QRS_NEXT_CUT()
PTP {E1 35817.312,E2 35817.312}
PTP {X 0,Y 759.87,A -85,B 0,C 180,E1 35817.312,E2 35817.312,E3 0,E4 0,E5 0,E6 0}
QRS_SPEED_INIT()
LIN {X 0,Y 759.87,Z 1164.5,A -85,B 0,C 180,E1 35817.312,E2 35817.312,E3 0,E4 0,E5 0,E6 0} C_VEL
LIN {X 0,Y 759.87,Z 412.653,A -85,B 0,C 180,E1 35817.312,E2 35817.312} C_VEL
LIN {X 0,Y 759.87,Z 404.575,A -85,B 0,C 180,E1 35817.312,E2 35817.312} C_VEL
LIN {X 0,Y 759.853,Z 402.575,A -85,B 0,C 180,E1 35817.162,E2 35817.162} C_VEL
LIN {X 0,Y 759.833,Z 402.574,A -85,B 0,C 180,E1 35814.715,E2 35814.715} C_VEL
LIN {X 0,Y 759.853,Z 402.572,A -85,B 0,C 180,E1 35812.255,E2 35812.255} C_VEL
LIN {X 0,Y 759.868,Z 402.576,A -85,B 0,C 180,E1 35809.231,E2 35809.231} C_VEL
LIN {X 0,Y 759.827,Z 402.575,A -85,B 0,C 180,E1 35806.763,E2 35806.763} C_VEL
LIN {X 0,Y 759.822,Z 402.575,A -85,B 0,C 180,E1 35804.506,E2 35804.506} C_VEL
LIN {X 0,Y 759.836,Z 402.574,A -85,B 0,C 180,E1 35802.145,E2 35802.145} C_VEL
LIN {X 0,Y 759.892,Z 402.577,A -85,B 0,C 180,E1 35799.27,E2 35799.27} C_VEL
LIN {X 0,Y 759.819,Z 402.576,A -85,B 0,C 180,E1 35796.665,E2 35796.665} C_VEL
LIN {X 0,Y 759.81,Z 402.576,A -85,B 0,C 180,E1 35794.428,E2 35794.428} C_VEL
LIN {X 0,Y 759.809,Z 402.576,A -85,B 0,C 180,E1 35792.234,E2 35792.234} C_VEL
LIN {X 0,Y 759.824,Z 402.577,A -85,B 0,C 180,E1 35789.909,E2 35789.909} C_VEL
LIN {X 0,Y 759.858,Z 402.577,A -85,B 0,C 180,E1 35786.953,E2 35786.953} C_VEL
LIN {X 0,Y 759.813,Z 402.576,A -85,B 0,C 180,E1 35784.525,E2 35784.525} C_VEL
LIN {X 0,Y 759.809,Z 402.577,A -85,B 0,C 180,E1 35782.366,E2 35782.366} C_VEL
LIN {X 0,Y 759.807,Z 402.577,A -85,B 0,C 180,E1 35780.223,E2 35780.223} C_VEL
LIN {X 0,Y 759.811,Z 402.576,A -85,B 0,C 180,E1 35778.033,E2 35778.033} C_VEL
LIN {X 0,Y 759.832,Z 402.577,A -85,B 0,C 180,E1 35775.672,E2 35775.672} C_VEL
LIN {X 0,Y 759.881,Z 402.574,A -85,B 0,C 180,E1 35772.756,E2 35772.756} C_VEL
LIN {X 0,Y 759.828,Z 402.575,A -85,B 0,C 180,E1 35770.248,E2 35770.248} C_VEL
LIN {X 0,Y 759.822,Z 402.575,A -85,B 0,C 180,E1 35767.919,E2 35767.919} C_VEL
LIN {X 0,Y 759.838,Z 402.576,A -85,B 0,C 180,E1 35765.566,E2 35765.566} C_VEL
LIN {X 0,Y 759.89,Z 402.904,A -85,B 0,C 180,E1 35765.147,E2 35765.147} C_VEL
LIN {X 0,Y 759.915,Z 438.12,A -85,B 0,C 180,E1 35762.827,E2 35762.827} C_VEL
LIN {X 0,Y 759.889,Z 482.271,A -85,B 0,C 180,E1 35760.023,E2 35760.023} C_VEL
LIN {X 0,Y 759.879,Z 498.982,A -85,B 0,C 180,E1 35758.995,E2 35758.995} C_VEL
LIN {X 0,Y 759.908,Z 754.621,A -85,B 0,C 180,E1 35756.312,E2 35756.312} C_VEL
LIN {X 0,Y 759.901,Z 846.139,A -85,B 0,C 180,E1 35755.349,E2 35755.349} C_VEL
LIN {X 0,Y 759.915,Z 869.708,A -85,B 0,C 180,E1 35754.962,E2 35754.962} C_VEL
LIN {X 0,Y 759.917,Z 889.343,A -85,B 0,C 180,E1 35754.528,E2 35754.528} C_VEL
LIN {X 0,Y 759.899,Z 912.803,A -85,B 0,C 180,E1 35753.865,E2 35753.865} C_VEL
LIN {X 0,Y 759.919,Z 931.783,A -85,B 0,C 180,E1 35753.209,E2 35753.209} C_VEL
LIN {X 0,Y 759.917,Z 953.84,A -85,B 0,C 180,E1 35752.3,E2 35752.3} C_VEL
LIN {X 0,Y 759.913,Z 972.967,A -85,B 0,C 180,E1 35751.375,E2 35751.375} C_VEL
LIN {X 0,Y 759.916,Z 992.86,A -85,B 0,C 180,E1 35750.255,E2 35750.255} C_VEL
LIN {X 0,Y 759.91,Z 1011.008,A -85,B 0,C 180,E1 35749.085,E2 35749.085} C_VEL
LIN {X 0,Y 759.908,Z 1028.563,A -85,B 0,C 180,E1 35747.774,E2 35747.774} C_VEL
LIN {X 0,Y 759.919,Z 1045.141,A -85,B 0,C 180,E1 35746.355,E2 35746.355} C_VEL
LIN {X 0,Y 759.902,Z 1059.575,A -85,B 0,C 180,E1 35744.946,E2 35744.946} C_VEL
LIN {X 0,Y 759.901,Z 1072.566,A -85,B 0,C 180,E1 35743.468,E2 35743.468} C_VEL
LIN {X 0,Y 759.915,Z 1084.432,A -85,B 0,C 180,E1 35741.922,E2 35741.922} C_VEL
LIN {X 0,Y 759.908,Z 1094.369,A -85,B 0,C 180,E1 35740.385,E2 35740.385} C_VEL
LIN {X 0,Y 759.894,Z 1103.565,A -85,B 0,C 180,E1 35738.703,E2 35738.703} C_VEL
LIN {X 0,Y 759.917,Z 1110.573,A -85,B 0,C 180,E1 35737.105,E2 35737.105} C_VEL
LIN {X 0,Y 759.896,Z 1116.604,A -85,B 0,C 180,E1 35735.361,E2 35735.361} C_VEL
LIN {X 0,Y 759.895,Z 1120.521,A -85,B 0,C 180,E1 35733.772,E2 35733.772} C_VEL
LIN {X 0,Y 759.915,Z 1123.316,A -85,B 0,C 180,E1 35732.036,E2 35732.036} C_VEL
LIN {X 0,Y 759.894,Z 1124.382,A -85,B 0,C 180,E1 35730.377,E2 35730.377} C_VEL
LIN {X 0,Y 759.893,Z 1123.929,A -85,B 0,C 180,E1 35728.567,E2 35728.567} C_VEL
LIN {X 0,Y 759.908,Z 1122.072,A -85,B 0,C 180,E1 35726.983,E2 35726.983} C_VEL
LIN {X 0,Y 759.892,Z 1118.285,A -85,B 0,C 180,E1 35725.169,E2 35725.169} C_VEL
LIN {X 0,Y 759.9,Z 1113.46,A -85,B 0,C 180,E1 35723.578,E2 35723.578} C_VEL
LIN {X 0,Y 759.912,Z 1106.463,A -85,B 0,C 180,E1 35721.83,E2 35721.83} C_VEL
LIN {X 0,Y 759.893,Z 1098.847,A -85,B 0,C 180,E1 35720.304,E2 35720.304} C_VEL
LIN {X 0,Y 759.9,Z 1088.594,A -85,B 0,C 180,E1 35718.605,E2 35718.605} C_VEL
LIN {X 0,Y 759.911,Z 1078.231,A -85,B 0,C 180,E1 35717.152,E2 35717.152} C_VEL
LIN {X 0,Y 759.917,Z 1065.021,A -85,B 0,C 180,E1 35715.564,E2 35715.564} C_VEL
LIN {X 0,Y 759.903,Z 1051.164,A -85,B 0,C 180,E1 35714.116,E2 35714.116} C_VEL
LIN {X 0,Y 759.905,Z 1035.427,A -85,B 0,C 180,E1 35712.7,E2 35712.7} C_VEL
LIN {X 0,Y 759.91,Z 1018.024,A -85,B 0,C 180,E1 35711.331,E2 35711.331} C_VEL
LIN {X 0,Y 759.91,Z 1000.339,A -85,B 0,C 180,E1 35710.115,E2 35710.115} C_VEL
LIN {X 0,Y 759.911,Z 981.35,A -85,B 0,C 180,E1 35708.988,E2 35708.988} C_VEL
LIN {X 0,Y 759.915,Z 961.832,A -85,B 0,C 180,E1 35707.976,E2 35707.976} C_VEL
LIN {X 0,Y 759.918,Z 941.464,A -85,B 0,C 180,E1 35707.081,E2 35707.081} C_VEL
LIN {X 0,Y 759.902,Z 920.345,A -85,B 0,C 180,E1 35706.289,E2 35706.289} C_VEL
LIN {X 0,Y 759.918,Z 899.782,A -85,B 0,C 180,E1 35705.659,E2 35705.659} C_VEL
LIN {X 0,Y 759.909,Z 878.291,A -85,B 0,C 180,E1 35705.119,E2 35705.119} C_VEL
LIN {X 0,Y 759.91,Z 857.163,A -85,B 0,C 180,E1 35704.725,E2 35704.725} C_VEL
LIN {X 0,Y 759.899,Z 835.535,A -85,B 0,C 180,E1 35704.431,E2 35704.431} C_VEL
LIN {X 0,Y 759.87,Z 588.613,A -85,B 0,C 180,E1 35701.868,E2 35701.868} C_VEL
LIN {X 0,Y 759.879,Z 498.825,A -85,B 0,C 180,E1 35700.91,E2 35700.91} C_VEL
LIN {X 0,Y 759.891,Z 459.664,A -85,B 0,C 180,E1 35698.461,E2 35698.461} C_VEL
LIN {X 0,Y 759.918,Z 417.942,A -85,B 0,C 180,E1 35695.771,E2 35695.771} C_VEL
LIN {X 0,Y 759.892,Z 402.857,A -85,B 0,C 180,E1 35694.756,E2 35694.756} C_VEL
LIN {X 0,Y 759.884,Z 402.572,A -85,B 0,C 180,E1 35693.386,E2 35693.386} C_VEL
LIN {X 0,Y 759.854,Z 402.576,A -85,B 0,C 180,E1 35690.439,E2 35690.439} C_VEL
LIN {X 0,Y 759.827,Z 402.575,A -85,B 0,C 180,E1 35688.031,E2 35688.031} C_VEL
LIN {X 0,Y 759.831,Z 402.573,A -85,B 0,C 180,E1 35685.672,E2 35685.672} C_VEL
LIN {X 0,Y 759.911,Z 402.574,A -85,B 0,C 180,E1 35682.968,E2 35682.968} C_VEL
LIN {X 0,Y 759.828,Z 402.576,A -85,B 0,C 180,E1 35680.132,E2 35680.132} C_VEL
LIN {X 0,Y 759.815,Z 402.576,A -85,B 0,C 180,E1 35677.853,E2 35677.853} C_VEL
LIN {X 0,Y 759.812,Z 402.575,A -85,B 0,C 180,E1 35675.66,E2 35675.66} C_VEL
LIN {X 0,Y 759.822,Z 402.576,A -85,B 0,C 180,E1 35673.372,E2 35673.372} C_VEL
LIN {X 0,Y 759.894,Z 402.578,A -85,B 0,C 180,E1 35670.525,E2 35670.525} C_VEL
LIN {X 0,Y 759.812,Z 402.577,A -85,B 0,C 180,E1 35667.936,E2 35667.936} C_VEL
LIN {X 0,Y 759.802,Z 402.577,A -85,B 0,C 180,E1 35665.65,E2 35665.65} C_VEL
LIN {X 0,Y 759.805,Z 402.577,A -85,B 0,C 180,E1 35663.5,E2 35663.5} C_VEL
LIN {X 0,Y 759.812,Z 402.577,A -85,B 0,C 180,E1 35661.297,E2 35661.297} C_VEL
LIN {X 0,Y 759.891,Z 402.577,A -85,B 0,C 180,E1 35658.648,E2 35658.648} C_VEL
LIN {X 0,Y 759.833,Z 402.575,A -85,B 0,C 180,E1 35655.807,E2 35655.807} C_VEL
LIN {X 0,Y 759.819,Z 402.575,A -85,B 0,C 180,E1 35653.468,E2 35653.468} C_VEL
LIN {X 0,Y 759.822,Z 402.575,A -85,B 0,C 180,E1 35651.231,E2 35651.231} C_VEL
LIN {X 0,Y 759.856,Z 402.576,A -85,B 0,C 180,E1 35648.78,E2 35648.78} C_VEL
LIN {X 0,Y 759.856,Z 402.573,A -85,B 0,C 180,E1 35645.74,E2 35645.74} C_VEL
LIN {X 0,Y 759.832,Z 402.573,A -85,B 0,C 180,E1 35643.319,E2 35643.319} C_VEL
LIN {X 0,Y 759.841,Z 402.575,A -85,B 0,C 180,E1 35640.905,E2 35640.905} C_VEL
LIN {X 0,Y 759.917,Z 402.575,A -85,B 0,C 180,E1 35638.19,E2 35638.19} C_VEL
LIN {X 0,Y 759.851,Z 402.571,A -85,B 0,C 180,E1 35635.396,E2 35635.396} C_VEL
LIN {X 0,Y 759.842,Z 402.573,A -85,B 0,C 180,E1 35632.97,E2 35632.97} C_VEL
LIN {X 0,Y 759.901,Z 402.577,A -85,B 0,C 180,E1 35630.304,E2 35630.304} C_VEL
LIN {X 0,Y 759.871,Z 402.569,A -85,B 0,C 180,E1 35627.383,E2 35627.383} C_VEL
LIN {X 0,Y 759.851,Z 402.573,A -85,B 0,C 180,E1 35624.819,E2 35624.819} C_VEL
LIN {X 0,Y 759.908,Z 402.578,A -85,B 0,C 180,E1 35622.147,E2 35622.147} C_VEL
LIN {X 0,Y 759.874,Z 402.569,A -85,B 0,C 180,E1 35619.189,E2 35619.189} C_VEL
LIN {X 0,Y 759.866,Z 402.573,A -85,B 0,C 180,E1 35616.516,E2 35616.516} C_VEL
LIN {X 0,Y 759.909,Z 402.572,A -85,B 0,C 180,E1 35613.761,E2 35613.761} C_VEL
LIN {X 0,Y 759.873,Z 402.568,A -85,B 0,C 180,E1 35610.951,E2 35610.951} C_VEL
LIN {X 0,Y 759.887,Z 402.575,A -85,B 0,C 180,E1 35608.216,E2 35608.216} C_VEL
LIN {X 0,Y 759.917,Z 402.564,A -85,B 0,C 180,E1 35605.268,E2 35605.268} C_VEL
LIN {X 0,Y 759.872,Z 402.572,A -85,B 0,C 180,E1 35602.465,E2 35602.465} C_VEL
LIN {X 0,Y 759.911,Z 402.575,A -85,B 0,C 180,E1 35599.744,E2 35599.744} C_VEL
LIN {X 0,Y 759.892,Z 402.566,A -85,B 0,C 180,E1 35596.801,E2 35596.801} C_VEL
LIN {X 0,Y 759.906,Z 402.576,A -85,B 0,C 180,E1 35593.903,E2 35593.903} C_VEL
LIN {X 0,Y 759.908,Z 402.565,A -85,B 0,C 180,E1 35590.835,E2 35590.835} C_VEL
LIN {X 0,Y 759.905,Z 402.577,A -85,B 0,C 180,E1 35587.862,E2 35587.862} C_VEL
LIN {X 0,Y 759.901,Z 402.734,A -85,B 0,C 180,E1 35585.893,E2 35585.893} C_VEL
LIN {X 0,Y 759.916,Z 406.955,A -85,B 0,C 180,E1 35585.594,E2 35585.594} C_VEL
LIN {X 0,Y 759.899,Z 450.794,A -85,B 0,C 180,E1 35582.913,E2 35582.913} C_VEL
LIN {X 0,Y 759.909,Z 452.682,A -85,B 0,C 180,E1 35582.815,E2 35582.815} C_VEL
LIN {X 0,Y 759.892,Z 704.216,A -85,B 0,C 180,E1 35580.08,E2 35580.08} C_VEL
LIN {X 0,Y 759.92,Z 841.979,A -85,B 0,C 180,E1 35578.595,E2 35578.595} C_VEL
LIN {X 0,Y 759.894,Z 866.292,A -85,B 0,C 180,E1 35578.211,E2 35578.211} C_VEL
LIN {X 0,Y 759.9,Z 887.681,A -85,B 0,C 180,E1 35577.742,E2 35577.742} C_VEL
LIN {X 0,Y 759.897,Z 907.094,A -85,B 0,C 180,E1 35577.221,E2 35577.221} C_VEL
LIN {X 0,Y 759.919,Z 929.734,A -85,B 0,C 180,E1 35576.491,E2 35576.491} C_VEL
LIN {X 0,Y 759.916,Z 951.248,A -85,B 0,C 180,E1 35575.652,E2 35575.652} C_VEL
LIN {X 0,Y 759.913,Z 970.659,A -85,B 0,C 180,E1 35574.783,E2 35574.783} C_VEL
LIN {X 0,Y 759.91,Z 993.058,A -85,B 0,C 180,E1 35573.62,E2 35573.62} C_VEL
LIN {X 0,Y 759.92,Z 1011.704,A -85,B 0,C 180,E1 35572.513,E2 35572.513} C_VEL
LIN {X 0,Y 759.906,Z 1031.522,A -85,B 0,C 180,E1 35571.173,E2 35571.173} C_VEL
LIN {X 0,Y 759.916,Z 1048.884,A -85,B 0,C 180,E1 35569.845,E2 35569.845} C_VEL
LIN {X 0,Y 759.917,Z 1065.39,A -85,B 0,C 180,E1 35568.409,E2 35568.409} C_VEL
LIN {X 0,Y 759.895,Z 1079.946,A -85,B 0,C 180,E1 35566.985,E2 35566.985} C_VEL
LIN {X 0,Y 759.899,Z 1094.876,A -85,B 0,C 180,E1 35565.312,E2 35565.312} C_VEL
LIN {X 0,Y 759.905,Z 1106.572,A -85,B 0,C 180,E1 35563.815,E2 35563.815} C_VEL
LIN {X 0,Y 759.9,Z 1118.785,A -85,B 0,C 180,E1 35561.999,E2 35561.999} C_VEL
LIN {X 0,Y 759.907,Z 1127.555,A -85,B 0,C 180,E1 35560.462,E2 35560.462} C_VEL
LIN {X 0,Y 759.888,Z 1136.073,A -85,B 0,C 180,E1 35558.704,E2 35558.704} C_VEL
LIN {X 0,Y 759.918,Z 1142.726,A -85,B 0,C 180,E1 35556.953,E2 35556.953} C_VEL
LIN {X 0,Y 759.883,Z 1147.51,A -85,B 0,C 180,E1 35555.361,E2 35555.361} C_VEL
LIN {X 0,Y 759.919,Z 1151.559,A -85,B 0,C 180,E1 35553.47,E2 35553.47} C_VEL
LIN {X 0,Y 759.902,Z 1153.63,A -85,B 0,C 180,E1 35551.81,E2 35551.81} C_VEL
LIN {X 0,Y 759.92,Z 1154.5,A -85,B 0,C 180,E1 35550,E2 35550} C_VEL
LIN {X 0,Y 759.902,Z 1153.63,A -85,B 0,C 180,E1 35548.19,E2 35548.19} C_VEL
LIN {X 0,Y 759.919,Z 1151.559,A -85,B 0,C 180,E1 35546.53,E2 35546.53} C_VEL
LIN {X 0,Y 759.883,Z 1147.51,A -85,B 0,C 180,E1 35544.639,E2 35544.639} C_VEL
LIN {X 0,Y 759.918,Z 1142.726,A -85,B 0,C 180,E1 35543.047,E2 35543.047} C_VEL
LIN {X 0,Y 759.889,Z 1135.729,A -85,B 0,C 180,E1 35541.22,E2 35541.22} C_VEL
LIN {X 0,Y 759.907,Z 1127.555,A -85,B 0,C 180,E1 35539.538,E2 35539.538} C_VEL
LIN {X 0,Y 759.9,Z 1118.785,A -85,B 0,C 180,E1 35538.001,E2 35538.001} C_VEL
LIN {X 0,Y 759.904,Z 1106.265,A -85,B 0,C 180,E1 35536.144,E2 35536.144} C_VEL
LIN {X 0,Y 759.9,Z 1094.679,A -85,B 0,C 180,E1 35534.664,E2 35534.664} C_VEL
LIN {X 0,Y 759.896,Z 1079.169,A -85,B 0,C 180,E1 35532.937,E2 35532.937} C_VEL
LIN {X 0,Y 759.914,Z 1064.539,A -85,B 0,C 180,E1 35531.512,E2 35531.512} C_VEL
LIN {X 0,Y 759.913,Z 1046.484,A -85,B 0,C 180,E1 35529.965,E2 35529.965} C_VEL
LIN {X 0,Y 759.91,Z 1029.578,A -85,B 0,C 180,E1 35528.684,E2 35528.684} C_VEL
LIN {X 0,Y 759.918,Z 1009.719,A -85,B 0,C 180,E1 35527.364,E2 35527.364} C_VEL
LIN {X 0,Y 759.91,Z 990.876,A -85,B 0,C 180,E1 35526.257,E2 35526.257} C_VEL
LIN {X 0,Y 759.913,Z 969.006,A -85,B 0,C 180,E1 35525.14,E2 35525.14} C_VEL
LIN {X 0,Y 759.917,Z 950.063,A -85,B 0,C 180,E1 35524.299,E2 35524.299} C_VEL
LIN {X 0,Y 759.915,Z 927.316,A -85,B 0,C 180,E1 35523.425,E2 35523.425} C_VEL
LIN {X 0,Y 759.899,Z 906.002,A -85,B 0,C 180,E1 35522.748,E2 35522.748} C_VEL
LIN {X 0,Y 759.898,Z 886.062,A -85,B 0,C 180,E1 35522.218,E2 35522.218} C_VEL
LIN {X 0,Y 759.898,Z 861.401,A -85,B 0,C 180,E1 35521.701,E2 35521.701} C_VEL
LIN {X 0,Y 759.92,Z 840.266,A -85,B 0,C 180,E1 35521.383,E2 35521.383} C_VEL
LIN {X 0,Y 759.859,Z 578.286,A -85,B 0,C 180,E1 35518.562,E2 35518.562} C_VEL
LIN {X 0,Y 759.907,Z 452.293,A -85,B 0,C 180,E1 35517.172,E2 35517.172} C_VEL
LIN {X 0,Y 759.92,Z 408.959,A -85,B 0,C 180,E1 35514.531,E2 35514.531} C_VEL
LIN {X 0,Y 759.902,Z 402.854,A -85,B 0,C 180,E1 35514.128,E2 35514.128} C_VEL
LIN {X 0,Y 759.903,Z 402.572,A -85,B 0,C 180,E1 35512.467,E2 35512.467} C_VEL
LIN {X 0,Y 759.882,Z 402.572,A -85,B 0,C 180,E1 35509.747,E2 35509.747} C_VEL
LIN {X 0,Y 759.909,Z 402.565,A -85,B 0,C 180,E1 35506.909,E2 35506.909} C_VEL
LIN {X 0,Y 759.896,Z 402.575,A -85,B 0,C 180,E1 35503.965,E2 35503.965} C_VEL
LIN {X 0,Y 759.9,Z 402.565,A -85,B 0,C 180,E1 35501.065,E2 35501.065} C_VEL
LIN {X 0,Y 759.908,Z 402.577,A -85,B 0,C 180,E1 35498.01,E2 35498.01} C_VEL
LIN {X 0,Y 759.877,Z 402.568,A -85,B 0,C 180,E1 35495.194,E2 35495.194} C_VEL
LIN {X 0,Y 759.906,Z 402.57,A -85,B 0,C 180,E1 35492.38,E2 35492.38} C_VEL
LIN {X 0,Y 759.873,Z 402.573,A -85,B 0,C 180,E1 35489.566,E2 35489.566} C_VEL
LIN {X 0,Y 759.888,Z 402.567,A -85,B 0,C 180,E1 35486.829,E2 35486.829} C_VEL
LIN {X 0,Y 759.901,Z 402.577,A -85,B 0,C 180,E1 35483.826,E2 35483.826} C_VEL
LIN {X 0,Y 759.859,Z 402.571,A -85,B 0,C 180,E1 35481.134,E2 35481.134} C_VEL
LIN {X 0,Y 759.912,Z 402.566,A -85,B 0,C 180,E1 35478.409,E2 35478.409} C_VEL
LIN {X 0,Y 759.873,Z 402.575,A -85,B 0,C 180,E1 35475.493,E2 35475.493} C_VEL
LIN {X 0,Y 759.852,Z 402.571,A -85,B 0,C 180,E1 35472.927,E2 35472.927} C_VEL
LIN {X 0,Y 759.917,Z 402.568,A -85,B 0,C 180,E1 35470.193,E2 35470.193} C_VEL
LIN {X 0,Y 759.863,Z 402.575,A -85,B 0,C 180,E1 35467.333,E2 35467.333} C_VEL
LIN {X 0,Y 759.844,Z 402.572,A -85,B 0,C 180,E1 35464.831,E2 35464.831} C_VEL
LIN {X 0,Y 759.895,Z 402.569,A -85,B 0,C 180,E1 35462.187,E2 35462.187} C_VEL
LIN {X 0,Y 759.86,Z 402.576,A -85,B 0,C 180,E1 35459.246,E2 35459.246} C_VEL
LIN {X 0,Y 759.853,Z 402.575,A -85,B 0,C 180,E1 35457.162,E2 35457.162} C_VEL
LIN {X 0,Y 758.828,Z 402.701,A -85,B 0,C 180,E1 35456.581,E2 35456.581} C_VEL
LIN {X 0,Y 752.415,Z 403.5,A -85,B 0,C 180,E1 35454.954,E2 35454.954} C_VEL
LIN {X 0,Y 751.899,Z 403.562,A -85,B 0,C 180,E1 35454.531,E2 35454.531} C_VEL
LIN {X 0,Y 751.971,Z 403.56,A -85,B 0,C 180,E1 35451.82,E2 35451.82} C_VEL
LIN {X 0,Y 751.9,Z 403.564,A -85,B 0,C 180,E1 35448.96,E2 35448.96} C_VEL
LIN {X 0,Y 751.885,Z 403.564,A -85,B 0,C 180,E1 35446.621,E2 35446.621} C_VEL
LIN {X 0,Y 751.89,Z 403.563,A -85,B 0,C 180,E1 35444.324,E2 35444.324} C_VEL
LIN {X 0,Y 751.977,Z 403.563,A -85,B 0,C 180,E1 35441.551,E2 35441.551} C_VEL
LIN {X 0,Y 751.888,Z 403.565,A -85,B 0,C 180,E1 35438.784,E2 35438.784} C_VEL
LIN {X 0,Y 751.874,Z 403.565,A -85,B 0,C 180,E1 35436.487,E2 35436.487} C_VEL
LIN {X 0,Y 751.872,Z 403.565,A -85,B 0,C 180,E1 35434.308,E2 35434.308} C_VEL
LIN {X 0,Y 751.883,Z 403.565,A -85,B 0,C 180,E1 35432.002,E2 35432.002} C_VEL
LIN {X 0,Y 751.958,Z 403.566,A -85,B 0,C 180,E1 35429.205,E2 35429.205} C_VEL
LIN {X 0,Y 751.87,Z 403.566,A -85,B 0,C 180,E1 35426.495,E2 35426.495} C_VEL
LIN {X 0,Y 751.865,Z 403.563,A -85,B 0,C 180,E1 35424.28,E2 35424.28} C_VEL
LIN {X 0,Y 751.869,Z 403.566,A -85,B 0,C 180,E1 35422.057,E2 35422.057} C_VEL
LIN {X 0,Y 751.888,Z 403.566,A -85,B 0,C 180,E1 35419.736,E2 35419.736} C_VEL
LIN {X 0,Y 751.93,Z 403.565,A -85,B 0,C 180,E1 35416.778,E2 35416.778} C_VEL
LIN {X 0,Y 751.882,Z 403.562,A -85,B 0,C 180,E1 35414.281,E2 35414.281} C_VEL
LIN {X 0,Y 751.879,Z 403.565,A -85,B 0,C 180,E1 35411.979,E2 35411.979} C_VEL
LIN {X 0,Y 751.901,Z 403.565,A -85,B 0,C 180,E1 35409.567,E2 35409.567} C_VEL
LIN {X 0,Y 751.95,Z 403.563,A -85,B 0,C 180,E1 35406.659,E2 35406.659} C_VEL
LIN {X 0,Y 751.93,Z 403.764,A -85,B 0,C 180,E1 35405.529,E2 35405.529} C_VEL
LIN {X 0,Y 752.835,Z 407.065,A -85,B 0,C 180,E1 35405.232,E2 35405.232} C_VEL
LIN {X 0,Y 752.698,Z 447.098,A -85,B 0,C 180,E1 35402.598,E2 35402.598} C_VEL
LIN {X 0,Y 752.547,Z 488.811,A -85,B 0,C 180,E1 35399.933,E2 35399.933} C_VEL
LIN {X 0,Y 752.641,Z 499.389,A -85,B 0,C 180,E1 35399.293,E2 35399.293} C_VEL
LIN {X 0,Y 752.884,Z 507.669,A -85,B 0,C 180,E1 35399.189,E2 35399.189} C_VEL
LIN {X 0,Y 752.725,Z 771.08,A -85,B 0,C 180,E1 35396.412,E2 35396.412} C_VEL
LIN {X 0,Y 752.664,Z 846.932,A -85,B 0,C 180,E1 35395.601,E2 35395.601} C_VEL
LIN {X 0,Y 752.63,Z 870.129,A -85,B 0,C 180,E1 35395.213,E2 35395.213} C_VEL
LIN {X 0,Y 752.589,Z 890.661,A -85,B 0,C 180,E1 35394.751,E2 35394.751} C_VEL
LIN {X 0,Y 752.497,Z 913.406,A -85,B 0,C 180,E1 35394.096,E2 35394.096} C_VEL
LIN {X 0,Y 752.459,Z 934.151,A -85,B 0,C 180,E1 35393.365,E2 35393.365} C_VEL
LIN {X 0,Y 752.373,Z 955.428,A -85,B 0,C 180,E1 35392.463,E2 35392.463} C_VEL
LIN {X 0,Y 752.305,Z 975.361,A -85,B 0,C 180,E1 35391.48,E2 35391.48} C_VEL
LIN {X 0,Y 752.229,Z 994.993,A -85,B 0,C 180,E1 35390.34,E2 35390.34} C_VEL
LIN {X 0,Y 752.153,Z 1014.194,A -85,B 0,C 180,E1 35389.058,E2 35389.058} C_VEL
LIN {X 0,Y 752.102,Z 1031.589,A -85,B 0,C 180,E1 35387.725,E2 35387.725} C_VEL
LIN {X 0,Y 752.051,Z 1047.695,A -85,B 0,C 180,E1 35386.292,E2 35386.292} C_VEL
LIN {X 0,Y 751.998,Z 1063.127,A -85,B 0,C 180,E1 35384.712,E2 35384.712} C_VEL
LIN {X 0,Y 751.962,Z 1076.4,A -85,B 0,C 180,E1 35383.143,E2 35383.143} C_VEL
LIN {X 0,Y 751.93,Z 1087.547,A -85,B 0,C 180,E1 35381.583,E2 35381.583} C_VEL
LIN {X 0,Y 751.922,Z 1097.557,A -85,B 0,C 180,E1 35379.955,E2 35379.955} C_VEL
LIN {X 0,Y 751.916,Z 1105.693,A -85,B 0,C 180,E1 35378.334,E2 35378.334} C_VEL
LIN {X 0,Y 751.893,Z 1112.824,A -85,B 0,C 180,E1 35376.592,E2 35376.592} C_VEL
LIN {X 0,Y 751.907,Z 1117.838,A -85,B 0,C 180,E1 35374.959,E2 35374.959} C_VEL
LIN {X 0,Y 751.903,Z 1121.716,A -85,B 0,C 180,E1 35373.202,E2 35373.202} C_VEL
LIN {X 0,Y 751.89,Z 1123.783,A -85,B 0,C 180,E1 35371.524,E2 35371.524} C_VEL
LIN {X 0,Y 751.903,Z 1124.453,A -85,B 0,C 180,E1 35369.771,E2 35369.771} C_VEL
LIN {X 0,Y 751.906,Z 1123.529,A -85,B 0,C 180,E1 35368.095,E2 35368.095} C_VEL
LIN {X 0,Y 751.895,Z 1120.867,A -85,B 0,C 180,E1 35366.264,E2 35366.264} C_VEL
LIN {X 0,Y 751.906,Z 1117.053,A -85,B 0,C 180,E1 35364.659,E2 35364.659} C_VEL
LIN {X 0,Y 751.915,Z 1110.93,A -85,B 0,C 180,E1 35362.819,E2 35362.819} C_VEL
LIN {X 0,Y 751.902,Z 1104.335,A -85,B 0,C 180,E1 35361.28,E2 35361.28} C_VEL
LIN {X 0,Y 751.924,Z 1094.909,A -85,B 0,C 180,E1 35359.503,E2 35359.503} C_VEL
LIN {X 0,Y 751.948,Z 1085.036,A -85,B 0,C 180,E1 35357.95,E2 35357.95} C_VEL
LIN {X 0,Y 751.966,Z 1073.307,A -85,B 0,C 180,E1 35356.387,E2 35356.387} C_VEL
LIN {X 0,Y 751.999,Z 1060.171,A -85,B 0,C 180,E1 35354.868,E2 35354.868} C_VEL
LIN {X 0,Y 752.049,Z 1045.259,A -85,B 0,C 180,E1 35353.39,E2 35353.39} C_VEL
LIN {X 0,Y 752.102,Z 1028.696,A -85,B 0,C 180,E1 35351.955,E2 35351.955} C_VEL
LIN {X 0,Y 752.155,Z 1011.697,A -85,B 0,C 180,E1 35350.67,E2 35350.67} C_VEL
LIN {X 0,Y 752.235,Z 993.152,A -85,B 0,C 180,E1 35349.457,E2 35349.457} C_VEL
LIN {X 0,Y 752.312,Z 973.943,A -85,B 0,C 180,E1 35348.357,E2 35348.357} C_VEL
LIN {X 0,Y 752.374,Z 954.701,A -85,B 0,C 180,E1 35347.414,E2 35347.414} C_VEL
LIN {X 0,Y 752.461,Z 933.111,A -85,B 0,C 180,E1 35346.506,E2 35346.506} C_VEL
LIN {X 0,Y 752.499,Z 912.966,A -85,B 0,C 180,E1 35345.8,E2 35345.8} C_VEL
LIN {X 0,Y 752.588,Z 889.081,A -85,B 0,C 180,E1 35345.12,E2 35345.12} C_VEL
LIN {X 0,Y 752.627,Z 868.915,A -85,B 0,C 180,E1 35344.673,E2 35344.673} C_VEL
LIN {X 0,Y 752.666,Z 844.6,A -85,B 0,C 180,E1 35344.28,E2 35344.28} C_VEL
LIN {X 0,Y 752.812,Z 584.295,A -85,B 0,C 180,E1 35341.535,E2 35341.535} C_VEL
LIN {X 0,Y 752.683,Z 499.611,A -85,B 0,C 180,E1 35340.622,E2 35340.622} C_VEL
LIN {X 0,Y 752.522,Z 495.177,A -85,B 0,C 180,E1 35340.377,E2 35340.377} C_VEL
LIN {X 0,Y 752.687,Z 454.668,A -85,B 0,C 180,E1 35337.802,E2 35337.802} C_VEL
LIN {X 0,Y 752.827,Z 413.061,A -85,B 0,C 180,E1 35335.079,E2 35335.079} C_VEL
LIN {X 0,Y 752.687,Z 406.102,A -85,B 0,C 180,E1 35334.606,E2 35334.606} C_VEL
LIN {X 0,Y 751.92,Z 403.665,A -85,B 0,C 180,E1 35334.356,E2 35334.356} C_VEL
LIN {X 0,Y 751.894,Z 403.562,A -85,B 0,C 180,E1 35331.899,E2 35331.899} C_VEL
LIN {X 0,Y 751.945,Z 403.561,A -85,B 0,C 180,E1 35329.284,E2 35329.284} C_VEL
LIN {X 0,Y 751.906,Z 403.563,A -85,B 0,C 180,E1 35326.337,E2 35326.337} C_VEL
LIN {X 0,Y 751.885,Z 403.565,A -85,B 0,C 180,E1 35323.962,E2 35323.962} C_VEL
LIN {X 0,Y 751.884,Z 403.563,A -85,B 0,C 180,E1 35321.636,E2 35321.636} C_VEL
LIN {X 0,Y 751.976,Z 403.563,A -85,B 0,C 180,E1 35318.874,E2 35318.874} C_VEL
LIN {X 0,Y 751.883,Z 403.563,A -85,B 0,C 180,E1 35316.045,E2 35316.045} C_VEL
LIN {X 0,Y 751.871,Z 403.566,A -85,B 0,C 180,E1 35313.772,E2 35313.772} C_VEL
LIN {X 0,Y 751.87,Z 403.565,A -85,B 0,C 180,E1 35311.51,E2 35311.51} C_VEL
LIN {X 0,Y 751.897,Z 403.566,A -85,B 0,C 180,E1 35309.109,E2 35309.109} C_VEL
LIN {X 0,Y 751.896,Z 403.566,A -85,B 0,C 180,E1 35306.115,E2 35306.115} C_VEL
LIN {X 0,Y 751.871,Z 403.566,A -85,B 0,C 180,E1 35303.763,E2 35303.763} C_VEL
LIN {X 0,Y 751.868,Z 403.566,A -85,B 0,C 180,E1 35301.534,E2 35301.534} C_VEL
LIN {X 0,Y 751.879,Z 403.566,A -85,B 0,C 180,E1 35299.23,E2 35299.23} C_VEL
LIN {X 0,Y 751.974,Z 403.566,A -85,B 0,C 180,E1 35296.453,E2 35296.453} C_VEL
LIN {X 0,Y 751.891,Z 403.563,A -85,B 0,C 180,E1 35293.693,E2 35293.693} C_VEL
LIN {X 0,Y 751.882,Z 403.564,A -85,B 0,C 180,E1 35291.351,E2 35291.351} C_VEL
LIN {X 0,Y 751.894,Z 403.565,A -85,B 0,C 180,E1 35289.028,E2 35289.028} C_VEL
LIN {X 0,Y 751.977,Z 403.562,A -85,B 0,C 180,E1 35286.183,E2 35286.183} C_VEL
LIN {X 0,Y 751.897,Z 403.561,A -85,B 0,C 180,E1 35283.431,E2 35283.431} C_VEL
LIN {X 0,Y 751.895,Z 403.563,A -85,B 0,C 180,E1 35281.067,E2 35281.067} C_VEL
LIN {X 0,Y 751.947,Z 403.564,A -85,B 0,C 180,E1 35278.476,E2 35278.476} C_VEL
LIN {X 0,Y 751.921,Z 403.559,A -85,B 0,C 180,E1 35275.5,E2 35275.5} C_VEL
LIN {X 0,Y 751.904,Z 403.562,A -85,B 0,C 180,E1 35272.973,E2 35272.973} C_VEL
LIN {X 0,Y 751.967,Z 403.566,A -85,B 0,C 180,E1 35270.278,E2 35270.278} C_VEL
LIN {X 0,Y 751.927,Z 403.559,A -85,B 0,C 180,E1 35267.325,E2 35267.325} C_VEL
LIN {X 0,Y 751.915,Z 403.562,A -85,B 0,C 180,E1 35264.734,E2 35264.734} C_VEL
LIN {X 0,Y 751.975,Z 403.562,A -85,B 0,C 180,E1 35261.952,E2 35261.952} C_VEL
LIN {X 0,Y 751.929,Z 403.558,A -85,B 0,C 180,E1 35259.122,E2 35259.122} C_VEL
LIN {X 0,Y 751.929,Z 403.563,A -85,B 0,C 180,E1 35256.489,E2 35256.489} C_VEL
LIN {X 0,Y 751.972,Z 403.559,A -85,B 0,C 180,E1 35253.633,E2 35253.633} C_VEL
LIN {X 0,Y 751.93,Z 403.558,A -85,B 0,C 180,E1 35250.876,E2 35250.876} C_VEL
LIN {X 0,Y 751.956,Z 403.565,A -85,B 0,C 180,E1 35248.136,E2 35248.136} C_VEL
LIN {X 0,Y 751.965,Z 403.553,A -85,B 0,C 180,E1 35245.126,E2 35245.126} C_VEL
LIN {X 0,Y 751.94,Z 403.563,A -85,B 0,C 180,E1 35242.288,E2 35242.288} C_VEL
LIN {X 0,Y 751.964,Z 403.56,A -85,B 0,C 180,E1 35239.517,E2 35239.517} C_VEL
LIN {X 0,Y 751.944,Z 403.556,A -85,B 0,C 180,E1 35236.667,E2 35236.667} C_VEL
LIN {X 0,Y 751.974,Z 403.565,A -85,B 0,C 180,E1 35233.778,E2 35233.778} C_VEL
LIN {X 0,Y 751.964,Z 403.555,A -85,B 0,C 180,E1 35230.76,E2 35230.76} C_VEL
LIN {X 0,Y 751.971,Z 403.565,A -85,B 0,C 180,E1 35227.806,E2 35227.806} C_VEL
LIN {X 0,Y 751.98,Z 403.796,A -85,B 0,C 180,E1 35226.255,E2 35226.255} C_VEL
LIN {X 0,Y 752.922,Z 406.722,A -85,B 0,C 180,E1 35225.99,E2 35225.99} C_VEL
LIN {X 0,Y 752.761,Z 449.219,A -85,B 0,C 180,E1 35223.361,E2 35223.361} C_VEL
LIN {X 0,Y 752.927,Z 453.168,A -85,B 0,C 180,E1 35223.15,E2 35223.15} C_VEL
LIN {X 0,Y 753.179,Z 459.277,A -85,B 0,C 180,E1 35223.066,E2 35223.066} C_VEL
LIN {X 0,Y 752.955,Z 714.779,A -85,B 0,C 180,E1 35220.272,E2 35220.272} C_VEL
LIN {X 0,Y 752.883,Z 842.408,A -85,B 0,C 180,E1 35218.882,E2 35218.882} C_VEL
LIN {X 0,Y 752.798,Z 867.202,A -85,B 0,C 180,E1 35218.482,E2 35218.482} C_VEL
LIN {X 0,Y 752.753,Z 888.593,A -85,B 0,C 180,E1 35218.006,E2 35218.006} C_VEL
LIN {X 0,Y 752.69,Z 909.676,A -85,B 0,C 180,E1 35217.428,E2 35217.428} C_VEL
LIN {X 0,Y 752.612,Z 934.071,A -85,B 0,C 180,E1 35216.604,E2 35216.604} C_VEL
LIN {X 0,Y 752.542,Z 953.239,A -85,B 0,C 180,E1 35215.837,E2 35215.837} C_VEL
LIN {X 0,Y 752.445,Z 975.244,A -85,B 0,C 180,E1 35214.822,E2 35214.822} C_VEL
LIN {X 0,Y 752.361,Z 995.242,A -85,B 0,C 180,E1 35213.746,E2 35213.746} C_VEL
LIN {X 0,Y 752.282,Z 1015.599,A -85,B 0,C 180,E1 35212.507,E2 35212.507} C_VEL
LIN {X 0,Y 752.195,Z 1034.285,A -85,B 0,C 180,E1 35211.197,E2 35211.197} C_VEL
LIN {X 0,Y 752.117,Z 1052.744,A -85,B 0,C 180,E1 35209.735,E2 35209.735} C_VEL
LIN {X 0,Y 752.079,Z 1068.793,A -85,B 0,C 180,E1 35208.286,E2 35208.286} C_VEL
LIN {X 0,Y 752.023,Z 1085.09,A -85,B 0,C 180,E1 35206.611,E2 35206.611} C_VEL
LIN {X 0,Y 751.972,Z 1097.889,A -85,B 0,C 180,E1 35205.107,E2 35205.107} C_VEL
LIN {X 0,Y 751.94,Z 1111.231,A -85,B 0,C 180,E1 35203.3,E2 35203.3} C_VEL
LIN {X 0,Y 751.929,Z 1120.637,A -85,B 0,C 180,E1 35201.817,E2 35201.817} C_VEL
LIN {X 0,Y 751.917,Z 1130.399,A -85,B 0,C 180,E1 35200.032,E2 35200.032} C_VEL
LIN {X 0,Y 751.918,Z 1138.205,A -85,B 0,C 180,E1 35198.257,E2 35198.257} C_VEL
LIN {X 0,Y 751.904,Z 1144.144,A -85,B 0,C 180,E1 35196.599,E2 35196.599} C_VEL
LIN {X 0,Y 751.915,Z 1149.336,A -85,B 0,C 180,E1 35194.653,E2 35194.653} C_VEL
LIN {X 0,Y 751.883,Z 1152.234,A -85,B 0,C 180,E1 35193.049,E2 35193.049} C_VEL
LIN {X 0,Y 751.913,Z 1154.149,A -85,B 0,C 180,E1 35191.219,E2 35191.219} C_VEL
LIN {X 0,Y 751.881,Z 1154.351,A -85,B 0,C 180,E1 35189.467,E2 35189.467} C_VEL
LIN {X 0,Y 751.919,Z 1153.296,A -85,B 0,C 180,E1 35187.79,E2 35187.79} C_VEL
LIN {X 0,Y 751.915,Z 1150.287,A -85,B 0,C 180,E1 35185.806,E2 35185.806} C_VEL
LIN {X 0,Y 751.918,Z 1146.481,A -85,B 0,C 180,E1 35184.2,E2 35184.2} C_VEL
LIN {X 0,Y 751.888,Z 1140.637,A -85,B 0,C 180,E1 35182.358,E2 35182.358} C_VEL
LIN {X 0,Y 751.921,Z 1133.519,A -85,B 0,C 180,E1 35180.646,E2 35180.646} C_VEL
LIN {X 0,Y 751.905,Z 1125.516,A -85,B 0,C 180,E1 35179.038,E2 35179.038} C_VEL
LIN {X 0,Y 751.937,Z 1114.349,A -85,B 0,C 180,E1 35177.169,E2 35177.169} C_VEL
LIN {X 0,Y 751.977,Z 1103.95,A -85,B 0,C 180,E1 35175.681,E2 35175.681} C_VEL
LIN {X 0,Y 752.003,Z 1090.042,A -85,B 0,C 180,E1 35173.945,E2 35173.945} C_VEL
LIN {X 0,Y 752.049,Z 1076.063,A -85,B 0,C 180,E1 35172.434,E2 35172.434} C_VEL
LIN {X 0,Y 752.114,Z 1059.246,A -85,B 0,C 180,E1 35170.83,E2 35170.83} C_VEL
LIN {X 0,Y 752.168,Z 1042.806,A -85,B 0,C 180,E1 35169.455,E2 35169.455} C_VEL
LIN {X 0,Y 752.246,Z 1022.85,A -85,B 0,C 180,E1 35167.986,E2 35167.986} C_VEL
LIN {X 0,Y 752.314,Z 1004.43,A -85,B 0,C 180,E1 35166.792,E2 35166.792} C_VEL
LIN {X 0,Y 752.417,Z 983.14,A -85,B 0,C 180,E1 35165.588,E2 35165.588} C_VEL
LIN {X 0,Y 752.491,Z 963.796,A -85,B 0,C 180,E1 35164.632,E2 35164.632} C_VEL
LIN {X 0,Y 752.602,Z 939.817,A -85,B 0,C 180,E1 35163.614,E2 35163.614} C_VEL
LIN {X 0,Y 752.649,Z 919.683,A -85,B 0,C 180,E1 35162.892,E2 35162.892} C_VEL
LIN {X 0,Y 752.749,Z 897.17,A -85,B 0,C 180,E1 35162.209,E2 35162.209} C_VEL
LIN {X 0,Y 752.785,Z 874.082,A -85,B 0,C 180,E1 35161.661,E2 35161.661} C_VEL
LIN {X 0,Y 752.845,Z 854.28,A -85,B 0,C 180,E1 35161.293,E2 35161.293} C_VEL
LIN {X 0,Y 752.889,Z 829.17,A -85,B 0,C 180,E1 35160.955,E2 35160.955} C_VEL
LIN {X 0,Y 753.025,Z 584.228,A -85,B 0,C 180,E1 35158.308,E2 35158.308} C_VEL
LIN {X 0,Y 753.004,Z 453.546,A -85,B 0,C 180,E1 35156.86,E2 35156.86} C_VEL
LIN {X 0,Y 752.762,Z 451.456,A -85,B 0,C 180,E1 35156.775,E2 35156.775} C_VEL
LIN {X 0,Y 752.922,Z 408.235,A -85,B 0,C 180,E1 35154.105,E2 35154.105} C_VEL
LIN {X 0,Y 752.649,Z 405.977,A -85,B 0,C 180,E1 35153.948,E2 35153.948} C_VEL
LIN {X 0,Y 751.958,Z 403.648,A -85,B 0,C 180,E1 35153.711,E2 35153.711} C_VEL
LIN {X 0,Y 751.964,Z 403.558,A -85,B 0,C 180,E1 35150.929,E2 35150.929} C_VEL
LIN {X 0,Y 751.958,Z 403.563,A -85,B 0,C 180,E1 35148.015,E2 35148.015} C_VEL
LIN {X 0,Y 751.97,Z 403.554,A -85,B 0,C 180,E1 35145.084,E2 35145.084} C_VEL
LIN {X 0,Y 751.973,Z 403.566,A -85,B 0,C 180,E1 35142.08,E2 35142.08} C_VEL
LIN {X 0,Y 751.946,Z 403.553,A -85,B 0,C 180,E1 35139.17,E2 35139.17} C_VEL
LIN {X 0,Y 751.969,Z 403.563,A -85,B 0,C 180,E1 35136.279,E2 35136.279} C_VEL
LIN {X 0,Y 751.932,Z 403.559,A -85,B 0,C 180,E1 35133.494,E2 35133.494} C_VEL
LIN {X 0,Y 751.975,Z 403.555,A -85,B 0,C 180,E1 35130.648,E2 35130.648} C_VEL
LIN {X 0,Y 751.943,Z 403.564,A -85,B 0,C 180,E1 35127.673,E2 35127.673} C_VEL
LIN {X 0,Y 751.937,Z 403.557,A -85,B 0,C 180,E1 35124.92,E2 35124.92} C_VEL
LIN {X 0,Y 751.975,Z 403.564,A -85,B 0,C 180,E1 35122.023,E2 35122.023} C_VEL
LIN {X 0,Y 751.92,Z 403.561,A -85,B 0,C 180,E1 35119.239,E2 35119.239} C_VEL
LIN {X 0,Y 751.957,Z 403.556,A -85,B 0,C 180,E1 35116.518,E2 35116.518} C_VEL
LIN {X 0,Y 751.939,Z 403.565,A -85,B 0,C 180,E1 35113.535,E2 35113.535} C_VEL
LIN {X 0,Y 751.91,Z 403.561,A -85,B 0,C 180,E1 35110.962,E2 35110.962} C_VEL
LIN {X 0,Y 751.956,Z 403.557,A -85,B 0,C 180,E1 35108.334,E2 35108.334} C_VEL
LIN {X 0,Y 751.927,Z 403.564,A -85,B 0,C 180,E1 35105.341,E2 35105.341} C_VEL
LIN {X 0,Y 751.903,Z 403.562,A -85,B 0,C 180,E1 35102.82,E2 35102.82} C_VEL
LIN {X 0,Y 751.942,Z 403.558,A -85,B 0,C 180,E1 35100.229,E2 35100.229} C_VEL
LIN {X 0,Y 751.924,Z 403.564,A -85,B 0,C 180,E1 35097.256,E2 35097.256} C_VEL
LIN {X 0,Y 751.894,Z 403.563,A -85,B 0,C 180,E1 35094.735,E2 35094.735} C_VEL
LIN {X 0,Y 751.899,Z 403.562,A -85,B 0,C 180,E1 35094.531,E2 35094.531} C_VEL
LIN {X 0,Y 750.928,Z 403.69,A -85,B 0,C 180,E1 35093.944,E2 35093.944} C_VEL
LIN {X 0,Y 744.537,Z 404.481,A -85,B 0,C 180,E1 35092.301,E2 35092.301} C_VEL
LIN {X 0,Y 744.028,Z 404.548,A -85,B 0,C 180,E1 35091.874,E2 35091.874} C_VEL
LIN {X 0,Y 743.964,Z 404.553,A -85,B 0,C 180,E1 35088.998,E2 35088.998} C_VEL
LIN {X 0,Y 743.947,Z 404.552,A -85,B 0,C 180,E1 35086.634,E2 35086.634} C_VEL
LIN {X 0,Y 743.951,Z 404.552,A -85,B 0,C 180,E1 35084.327,E2 35084.327} C_VEL
LIN {X 0,Y 744.033,Z 404.552,A -85,B 0,C 180,E1 35081.583,E2 35081.583} C_VEL
LIN {X 0,Y 743.951,Z 404.554,A -85,B 0,C 180,E1 35078.805,E2 35078.805} C_VEL
LIN {X 0,Y 743.936,Z 404.554,A -85,B 0,C 180,E1 35076.473,E2 35076.473} C_VEL
LIN {X 0,Y 743.937,Z 404.554,A -85,B 0,C 180,E1 35074.184,E2 35074.184} C_VEL
LIN {X 0,Y 743.996,Z 404.554,A -85,B 0,C 180,E1 35071.591,E2 35071.591} C_VEL
LIN {X 0,Y 743.949,Z 404.555,A -85,B 0,C 180,E1 35068.739,E2 35068.739} C_VEL
LIN {X 0,Y 743.927,Z 404.556,A -85,B 0,C 180,E1 35066.375,E2 35066.375} C_VEL
LIN {X 0,Y 743.927,Z 404.55,A -85,B 0,C 180,E1 35064.125,E2 35064.125} C_VEL
LIN {X 0,Y 743.944,Z 404.555,A -85,B 0,C 180,E1 35061.811,E2 35061.811} C_VEL
LIN {X 0,Y 744.005,Z 404.551,A -85,B 0,C 180,E1 35058.914,E2 35058.914} C_VEL
LIN {X 0,Y 743.941,Z 404.555,A -85,B 0,C 180,E1 35056.303,E2 35056.303} C_VEL
LIN {X 0,Y 743.938,Z 404.551,A -85,B 0,C 180,E1 35054.018,E2 35054.018} C_VEL
LIN {X 0,Y 743.96,Z 404.556,A -85,B 0,C 180,E1 35051.601,E2 35051.601} C_VEL
LIN {X 0,Y 744.003,Z 404.551,A -85,B 0,C 180,E1 35048.663,E2 35048.663} C_VEL
LIN {X 0,Y 743.95,Z 404.555,A -85,B 0,C 180,E1 35046.064,E2 35046.064} C_VEL
LIN {X 0,Y 744.032,Z 405.084,A -85,B 0,C 180,E1 35045.855,E2 35045.855} C_VEL
LIN {X 0,Y 745.777,Z 410.332,A -85,B 0,C 180,E1 35045.394,E2 35045.394} C_VEL
LIN {X 0,Y 745.501,Z 450.652,A -85,B 0,C 180,E1 35042.719,E2 35042.719} C_VEL
LIN {X 0,Y 745.238,Z 490.975,A -85,B 0,C 180,E1 35040.119,E2 35040.119} C_VEL
LIN {X 0,Y 745.284,Z 499.252,A -85,B 0,C 180,E1 35039.614,E2 35039.614} C_VEL
LIN {X 0,Y 745.897,Z 503.596,A -85,B 0,C 180,E1 35039.534,E2 35039.534} C_VEL
LIN {X 0,Y 745.563,Z 767.339,A -85,B 0,C 180,E1 35036.725,E2 35036.725} C_VEL
LIN {X 0,Y 745.444,Z 846.868,A -85,B 0,C 180,E1 35035.869,E2 35035.869} C_VEL
LIN {X 0,Y 745.36,Z 870.263,A -85,B 0,C 180,E1 35035.474,E2 35035.474} C_VEL
LIN {X 0,Y 745.275,Z 891.225,A -85,B 0,C 180,E1 35034.997,E2 35034.997} C_VEL
LIN {X 0,Y 745.109,Z 914.004,A -85,B 0,C 180,E1 35034.331,E2 35034.331} C_VEL
LIN {X 0,Y 745.006,Z 935.7,A -85,B 0,C 180,E1 35033.555,E2 35033.555} C_VEL
LIN {X 0,Y 744.838,Z 956.333,A -85,B 0,C 180,E1 35032.661,E2 35032.661} C_VEL
LIN {X 0,Y 744.683,Z 976.838,A -85,B 0,C 180,E1 35031.628,E2 35031.628} C_VEL
LIN {X 0,Y 744.55,Z 995.665,A -85,B 0,C 180,E1 35030.519,E2 35030.519} C_VEL
LIN {X 0,Y 744.394,Z 1014.89,A -85,B 0,C 180,E1 35029.214,E2 35029.214} C_VEL
LIN {X 0,Y 744.293,Z 1031.595,A -85,B 0,C 180,E1 35027.917,E2 35027.917} C_VEL
LIN {X 0,Y 744.19,Z 1047.701,A -85,B 0,C 180,E1 35026.469,E2 35026.469} C_VEL
LIN {X 0,Y 744.083,Z 1063.132,A -85,B 0,C 180,E1 35024.872,E2 35024.872} C_VEL
LIN {X 0,Y 744.022,Z 1076.404,A -85,B 0,C 180,E1 35023.286,E2 35023.286} C_VEL
LIN {X 0,Y 743.969,Z 1087.552,A -85,B 0,C 180,E1 35021.709,E2 35021.709} C_VEL
LIN {X 0,Y 743.951,Z 1097.561,A -85,B 0,C 180,E1 35020.063,E2 35020.063} C_VEL
LIN {X 0,Y 743.922,Z 1105.764,A -85,B 0,C 180,E1 35018.409,E2 35018.409} C_VEL
LIN {X 0,Y 743.9,Z 1112.655,A -85,B 0,C 180,E1 35016.715,E2 35016.715} C_VEL
LIN {X 0,Y 743.911,Z 1117.84,A -85,B 0,C 180,E1 35015.012,E2 35015.012} C_VEL
LIN {X 0,Y 743.9,Z 1121.716,A -85,B 0,C 180,E1 35013.236,E2 35013.236} C_VEL
LIN {X 0,Y 743.89,Z 1123.784,A -85,B 0,C 180,E1 35011.54,E2 35011.54} C_VEL
LIN {X 0,Y 743.903,Z 1124.452,A -85,B 0,C 180,E1 35009.769,E2 35009.769} C_VEL
LIN {X 0,Y 743.908,Z 1123.529,A -85,B 0,C 180,E1 35008.074,E2 35008.074} C_VEL
LIN {X 0,Y 743.897,Z 1120.866,A -85,B 0,C 180,E1 35006.224,E2 35006.224} C_VEL
LIN {X 0,Y 743.905,Z 1117.052,A -85,B 0,C 180,E1 35004.601,E2 35004.601} C_VEL
LIN {X 0,Y 743.923,Z 1110.838,A -85,B 0,C 180,E1 35002.718,E2 35002.718} C_VEL
LIN {X 0,Y 743.916,Z 1103.979,A -85,B 0,C 180,E1 35001.108,E2 35001.108} C_VEL
LIN {X 0,Y 743.945,Z 1094.907,A -85,B 0,C 180,E1 34999.389,E2 34999.389} C_VEL
LIN {X 0,Y 743.994,Z 1085.033,A -85,B 0,C 180,E1 34997.819,E2 34997.819} C_VEL
LIN {X 0,Y 744.038,Z 1073.304,A -85,B 0,C 180,E1 34996.239,E2 34996.239} C_VEL
LIN {X 0,Y 744.101,Z 1060.398,A -85,B 0,C 180,E1 34994.729,E2 34994.729} C_VEL
LIN {X 0,Y 744.188,Z 1046.104,A -85,B 0,C 180,E1 34993.29,E2 34993.29} C_VEL
LIN {X 0,Y 744.298,Z 1030.226,A -85,B 0,C 180,E1 34991.882,E2 34991.882} C_VEL
LIN {X 0,Y 744.402,Z 1012.927,A -85,B 0,C 180,E1 34990.551,E2 34990.551} C_VEL
LIN {X 0,Y 744.557,Z 993.808,A -85,B 0,C 180,E1 34989.276,E2 34989.276} C_VEL
LIN {X 0,Y 744.719,Z 974.737,A -85,B 0,C 180,E1 34988.166,E2 34988.166} C_VEL
LIN {X 0,Y 744.845,Z 954.694,A -85,B 0,C 180,E1 34987.172,E2 34987.172} C_VEL
LIN {X 0,Y 745.018,Z 932.937,A -85,B 0,C 180,E1 34986.251,E2 34986.251} C_VEL
LIN {X 0,Y 745.113,Z 912.954,A -85,B 0,C 180,E1 34985.544,E2 34985.544} C_VEL
LIN {X 0,Y 745.276,Z 888.955,A -85,B 0,C 180,E1 34984.857,E2 34984.857} C_VEL
LIN {X 0,Y 745.36,Z 868.381,A -85,B 0,C 180,E1 34984.397,E2 34984.397} C_VEL
LIN {X 0,Y 745.447,Z 844.32,A -85,B 0,C 180,E1 34984.009,E2 34984.009} C_VEL
LIN {X 0,Y 745.769,Z 585.701,A -85,B 0,C 180,E1 34981.257,E2 34981.257} C_VEL
LIN {X 0,Y 745.694,Z 501.172,A -85,B 0,C 180,E1 34980.34,E2 34980.34} C_VEL
LIN {X 0,Y 745.217,Z 498.68,A -85,B 0,C 180,E1 34980.275,E2 34980.275} C_VEL
LIN {X 0,Y 745.476,Z 458.029,A -85,B 0,C 180,E1 34977.673,E2 34977.673} C_VEL
LIN {X 0,Y 745.745,Z 415.836,A -85,B 0,C 180,E1 34974.886,E2 34974.886} C_VEL
LIN {X 0,Y 745.734,Z 409.791,A -85,B 0,C 180,E1 34974.477,E2 34974.477} C_VEL
LIN {X 0,Y 743.982,Z 404.736,A -85,B 0,C 180,E1 34974.006,E2 34974.006} C_VEL
LIN {X 0,Y 743.981,Z 404.55,A -85,B 0,C 180,E1 34971.518,E2 34971.518} C_VEL
LIN {X 0,Y 743.981,Z 404.556,A -85,B 0,C 180,E1 34968.469,E2 34968.469} C_VEL
LIN {X 0,Y 743.947,Z 404.55,A -85,B 0,C 180,E1 34965.977,E2 34965.977} C_VEL
LIN {X 0,Y 743.949,Z 404.554,A -85,B 0,C 180,E1 34963.69,E2 34963.69} C_VEL
LIN {X 0,Y 744.022,Z 404.549,A -85,B 0,C 180,E1 34960.982,E2 34960.982} C_VEL
LIN {X 0,Y 743.954,Z 404.555,A -85,B 0,C 180,E1 34958.163,E2 34958.163} C_VEL
LIN {X 0,Y 743.936,Z 404.55,A -85,B 0,C 180,E1 34955.858,E2 34955.858} C_VEL
LIN {X 0,Y 743.933,Z 404.555,A -85,B 0,C 180,E1 34953.625,E2 34953.625} C_VEL
LIN {X 0,Y 743.958,Z 404.554,A -85,B 0,C 180,E1 34951.161,E2 34951.161} C_VEL
LIN {X 0,Y 743.956,Z 404.555,A -85,B 0,C 180,E1 34948.148,E2 34948.148} C_VEL
LIN {X 0,Y 743.927,Z 404.555,A -85,B 0,C 180,E1 34945.73,E2 34945.73} C_VEL
LIN {X 0,Y 743.928,Z 404.555,A -85,B 0,C 180,E1 34943.528,E2 34943.528} C_VEL
LIN {X 0,Y 743.937,Z 404.554,A -85,B 0,C 180,E1 34941.278,E2 34941.278} C_VEL
LIN {X 0,Y 744.034,Z 404.555,A -85,B 0,C 180,E1 34938.491,E2 34938.491} C_VEL
LIN {X 0,Y 743.946,Z 404.553,A -85,B 0,C 180,E1 34935.673,E2 34935.673} C_VEL
LIN {X 0,Y 743.941,Z 404.553,A -85,B 0,C 180,E1 34933.366,E2 34933.366} C_VEL
LIN {X 0,Y 743.957,Z 404.554,A -85,B 0,C 180,E1 34931.002,E2 34931.002} C_VEL
LIN {X 0,Y 744.026,Z 404.549,A -85,B 0,C 180,E1 34928.112,E2 34928.112} C_VEL
LIN {X 0,Y 743.953,Z 404.552,A -85,B 0,C 180,E1 34925.398,E2 34925.398} C_VEL
LIN {X 0,Y 743.958,Z 404.551,A -85,B 0,C 180,E1 34923.005,E2 34923.005} C_VEL
LIN {X 0,Y 744.038,Z 404.552,A -85,B 0,C 180,E1 34920.231,E2 34920.231} C_VEL
LIN {X 0,Y 743.969,Z 404.55,A -85,B 0,C 180,E1 34917.381,E2 34917.381} C_VEL
LIN {X 0,Y 743.965,Z 404.551,A -85,B 0,C 180,E1 34914.911,E2 34914.911} C_VEL
LIN {X 0,Y 744.041,Z 404.554,A -85,B 0,C 180,E1 34912.199,E2 34912.199} C_VEL
LIN {X 0,Y 743.982,Z 404.548,A -85,B 0,C 180,E1 34909.312,E2 34909.312} C_VEL
LIN {X 0,Y 743.977,Z 404.552,A -85,B 0,C 180,E1 34906.713,E2 34906.713} C_VEL
LIN {X 0,Y 744.035,Z 404.551,A -85,B 0,C 180,E1 34903.92,E2 34903.92} C_VEL
LIN {X 0,Y 743.985,Z 404.547,A -85,B 0,C 180,E1 34901.101,E2 34901.101} C_VEL
LIN {X 0,Y 743.995,Z 404.552,A -85,B 0,C 180,E1 34898.438,E2 34898.438} C_VEL
LIN {X 0,Y 744.039,Z 404.544,A -85,B 0,C 180,E1 34895.464,E2 34895.464} C_VEL
LIN {X 0,Y 743.985,Z 404.55,A -85,B 0,C 180,E1 34892.669,E2 34892.669} C_VEL
LIN {X 0,Y 744.038,Z 404.555,A -85,B 0,C 180,E1 34889.916,E2 34889.916} C_VEL
LIN {X 0,Y 744.003,Z 404.543,A -85,B 0,C 180,E1 34886.932,E2 34886.932} C_VEL
LIN {X 0,Y 744.015,Z 404.552,A -85,B 0,C 180,E1 34884.13,E2 34884.13} C_VEL
LIN {X 0,Y 744.034,Z 404.538,A -85,B 0,C 180,E1 34881.088,E2 34881.088} C_VEL
LIN {X 0,Y 744.006,Z 404.552,A -85,B 0,C 180,E1 34878.195,E2 34878.195} C_VEL
LIN {X 0,Y 744.024,Z 404.547,A -85,B 0,C 180,E1 34875.31,E2 34875.31} C_VEL
LIN {X 0,Y 744.006,Z 404.544,A -85,B 0,C 180,E1 34872.532,E2 34872.532} C_VEL
LIN {X 0,Y 744.032,Z 404.55,A -85,B 0,C 180,E1 34869.642,E2 34869.642} C_VEL
LIN {X 0,Y 744.044,Z 404.68,A -85,B 0,C 180,E1 34866.659,E2 34866.659} C_VEL
LIN {X 0,Y 745.522,Z 408.959,A -85,B 0,C 180,E1 34866.261,E2 34866.261} C_VEL
LIN {X 0,Y 745.938,Z 411.196,A -85,B 0,C 180,E1 34866.095,E2 34866.095} C_VEL
LIN {X 0,Y 745.724,Z 452.732,A -85,B 0,C 180,E1 34863.519,E2 34863.519} C_VEL
LIN {X 0,Y 746.468,Z 457.229,A -85,B 0,C 180,E1 34863.425,E2 34863.425} C_VEL
LIN {X 0,Y 746.041,Z 713.379,A -85,B 0,C 180,E1 34860.598,E2 34860.598} C_VEL
LIN {X 0,Y 745.867,Z 842.515,A -85,B 0,C 180,E1 34859.179,E2 34859.179} C_VEL
LIN {X 0,Y 745.721,Z 867.473,A -85,B 0,C 180,E1 34858.771,E2 34858.771} C_VEL
LIN {X 0,Y 745.622,Z 888.919,A -85,B 0,C 180,E1 34858.289,E2 34858.289} C_VEL
LIN {X 0,Y 745.498,Z 911.074,A -85,B 0,C 180,E1 34857.674,E2 34857.674} C_VEL
LIN {X 0,Y 745.321,Z 934.807,A -85,B 0,C 180,E1 34856.857,E2 34856.857} C_VEL
LIN {X 0,Y 745.177,Z 955.231,A -85,B 0,C 180,E1 34856.026,E2 34856.026} C_VEL
LIN {X 0,Y 744.964,Z 978.331,A -85,B 0,C 180,E1 34854.926,E2 34854.926} C_VEL
LIN {X 0,Y 744.817,Z 997.354,A -85,B 0,C 180,E1 34853.88,E2 34853.88} C_VEL
LIN {X 0,Y 744.62,Z 1019.23,A -85,B 0,C 180,E1 34852.501,E2 34852.501} C_VEL
LIN {X 0,Y 744.487,Z 1036.823,A -85,B 0,C 180,E1 34851.237,E2 34851.237} C_VEL
LIN {X 0,Y 744.33,Z 1054.602,A -85,B 0,C 180,E1 34849.787,E2 34849.787} C_VEL
LIN {X 0,Y 744.242,Z 1070.494,A -85,B 0,C 180,E1 34848.323,E2 34848.323} C_VEL
LIN {X 0,Y 744.131,Z 1085.799,A -85,B 0,C 180,E1 34846.712,E2 34846.712} C_VEL
LIN {X 0,Y 744.053,Z 1098.533,A -85,B 0,C 180,E1 34845.192,E2 34845.192} C_VEL
LIN {X 0,Y 743.987,Z 1111.752,A -85,B 0,C 180,E1 34843.366,E2 34843.366} C_VEL
LIN {X 0,Y 743.958,Z 1121.101,A -85,B 0,C 180,E1 34841.867,E2 34841.867} C_VEL
LIN {X 0,Y 743.934,Z 1130.759,A -85,B 0,C 180,E1 34840.063,E2 34840.063} C_VEL
LIN {X 0,Y 743.918,Z 1138.206,A -85,B 0,C 180,E1 34838.347,E2 34838.347} C_VEL
LIN {X 0,Y 743.91,Z 1143.997,A -85,B 0,C 180,E1 34836.715,E2 34836.715} C_VEL
LIN {X 0,Y 743.902,Z 1149.178,A -85,B 0,C 180,E1 34834.78,E2 34834.78} C_VEL
LIN {X 0,Y 743.89,Z 1152.121,A -85,B 0,C 180,E1 34833.159,E2 34833.159} C_VEL
LIN {X 0,Y 743.901,Z 1154.032,A -85,B 0,C 180,E1 34831.386,E2 34831.386} C_VEL
LIN {X 0,Y 743.883,Z 1154.373,A -85,B 0,C 180,E1 34829.538,E2 34829.538} C_VEL
LIN {X 0,Y 743.916,Z 1153.43,A -85,B 0,C 180,E1 34827.92,E2 34827.92} C_VEL
LIN {X 0,Y 743.916,Z 1150.605,A -85,B 0,C 180,E1 34825.915,E2 34825.915} C_VEL
LIN {X 0,Y 743.918,Z 1146.687,A -85,B 0,C 180,E1 34824.214,E2 34824.214} C_VEL
LIN {X 0,Y 743.891,Z 1141.2,A -85,B 0,C 180,E1 34822.431,E2 34822.431} C_VEL
LIN {X 0,Y 743.929,Z 1133.737,A -85,B 0,C 180,E1 34820.592,E2 34820.592} C_VEL
LIN {X 0,Y 743.926,Z 1126.333,A -85,B 0,C 180,E1 34819.075,E2 34819.075} C_VEL
LIN {X 0,Y 743.986,Z 1115.909,A -85,B 0,C 180,E1 34817.267,E2 34817.267} C_VEL
LIN {X 0,Y 744.036,Z 1105.097,A -85,B 0,C 180,E1 34815.682,E2 34815.682} C_VEL
LIN {X 0,Y 744.099,Z 1092.116,A -85,B 0,C 180,E1 34814.01,E2 34814.01} C_VEL
LIN {X 0,Y 744.189,Z 1077.619,A -85,B 0,C 180,E1 34812.404,E2 34812.404} C_VEL
LIN {X 0,Y 744.304,Z 1061.99,A -85,B 0,C 180,E1 34810.865,E2 34810.865} C_VEL
LIN {X 0,Y 744.42,Z 1044.831,A -85,B 0,C 180,E1 34809.396,E2 34809.396} C_VEL
LIN {X 0,Y 744.579,Z 1026.474,A -85,B 0,C 180,E1 34807.996,E2 34807.996} C_VEL
LIN {X 0,Y 744.717,Z 1007.739,A -85,B 0,C 180,E1 34806.75,E2 34806.75} C_VEL
LIN {X 0,Y 744.922,Z 987.074,A -85,B 0,C 180,E1 34805.533,E2 34805.533} C_VEL
LIN {X 0,Y 745.071,Z 966.344,A -85,B 0,C 180,E1 34804.483,E2 34804.483} C_VEL
LIN {X 0,Y 745.278,Z 944.262,A -85,B 0,C 180,E1 34803.507,E2 34803.507} C_VEL
LIN {X 0,Y 745.41,Z 921.533,A -85,B 0,C 180,E1 34802.669,E2 34802.669} C_VEL
LIN {X 0,Y 745.547,Z 900.872,A -85,B 0,C 180,E1 34802.026,E2 34802.026} C_VEL
LIN {X 0,Y 745.695,Z 875.926,A -85,B 0,C 180,E1 34801.406,E2 34801.406} C_VEL
LIN {X 0,Y 745.798,Z 855.578,A -85,B 0,C 180,E1 34801.018,E2 34801.018} C_VEL
LIN {X 0,Y 745.883,Z 832.129,A -85,B 0,C 180,E1 34800.689,E2 34800.689} C_VEL
LIN {X 0,Y 746.21,Z 585.475,A -85,B 0,C 180,E1 34797.999,E2 34797.999} C_VEL
LIN {X 0,Y 746.287,Z 455.193,A -85,B 0,C 180,E1 34796.542,E2 34796.542} C_VEL
LIN {X 0,Y 745.667,Z 452.278,A -85,B 0,C 180,E1 34796.463,E2 34796.463} C_VEL
LIN {X 0,Y 745.942,Z 410.45,A -85,B 0,C 180,E1 34793.857,E2 34793.857} C_VEL
LIN {X 0,Y 744.048,Z 404.712,A -85,B 0,C 180,E1 34793.349,E2 34793.349} C_VEL
LIN {X 0,Y 744.027,Z 404.55,A -85,B 0,C 180,E1 34790.431,E2 34790.431} C_VEL
LIN {X 0,Y 744.003,Z 404.546,A -85,B 0,C 180,E1 34787.572,E2 34787.572} C_VEL
LIN {X 0,Y 744.027,Z 404.546,A -85,B 0,C 180,E1 34784.765,E2 34784.765} C_VEL
LIN {X 0,Y 744.013,Z 404.553,A -85,B 0,C 180,E1 34781.881,E2 34781.881} C_VEL
LIN {X 0,Y 744.019,Z 404.539,A -85,B 0,C 180,E1 34779.033,E2 34779.033} C_VEL
LIN {X 0,Y 744.027,Z 404.553,A -85,B 0,C 180,E1 34775.964,E2 34775.964} C_VEL
LIN {X 0,Y 743.999,Z 404.543,A -85,B 0,C 180,E1 34773.146,E2 34773.146} C_VEL
LIN {X 0,Y 744.03,Z 404.551,A -85,B 0,C 180,E1 34770.262,E2 34770.262} C_VEL
LIN {X 0,Y 743.99,Z 404.551,A -85,B 0,C 180,E1 34767.45,E2 34767.45} C_VEL
LIN {X 0,Y 744.019,Z 404.544,A -85,B 0,C 180,E1 34764.703,E2 34764.703} C_VEL
LIN {X 0,Y 744.012,Z 404.553,A -85,B 0,C 180,E1 34761.69,E2 34761.69} C_VEL
LIN {X 0,Y 743.983,Z 404.547,A -85,B 0,C 180,E1 34758.98,E2 34758.98} C_VEL
LIN {X 0,Y 744.035,Z 404.548,A -85,B 0,C 180,E1 34756.152,E2 34756.152} C_VEL
LIN {X 0,Y 743.982,Z 404.552,A -85,B 0,C 180,E1 34753.335,E2 34753.335} C_VEL
LIN {X 0,Y 743.98,Z 404.548,A -85,B 0,C 180,E1 34750.75,E2 34750.75} C_VEL
LIN {X 0,Y 744.039,Z 404.552,A -85,B 0,C 180,E1 34747.879,E2 34747.879} C_VEL
LIN {X 0,Y 743.971,Z 404.551,A -85,B 0,C 180,E1 34745.089,E2 34745.089} C_VEL
LIN {X 0,Y 743.977,Z 404.549,A -85,B 0,C 180,E1 34742.542,E2 34742.542} C_VEL
LIN {X 0,Y 744.032,Z 404.556,A -85,B 0,C 180,E1 34739.615,E2 34739.615} C_VEL
LIN {X 0,Y 743.96,Z 404.551,A -85,B 0,C 180,E1 34736.918,E2 34736.918} C_VEL
LIN {X 0,Y 743.961,Z 404.551,A -85,B 0,C 180,E1 34734.524,E2 34734.524} C_VEL
LIN {X 0,Y 744.028,Z 404.548,A -85,B 0,C 180,E1 34731.874,E2 34731.874} C_VEL
LIN {X 0,Y 743.074,Z 404.677,A -85,B 0,C 180,E1 34731.281,E2 34731.281} C_VEL
LIN {X 0,Y 736.626,Z 405.479,A -85,B 0,C 180,E1 34729.621,E2 34729.621} C_VEL
LIN {X 0,Y 736.047,Z 405.543,A -85,B 0,C 180,E1 34729.189,E2 34729.189} C_VEL
LIN {X 0,Y 736.011,Z 405.542,A -85,B 0,C 180,E1 34726.727,E2 34726.727} C_VEL
LIN {X 0,Y 736.01,Z 405.542,A -85,B 0,C 180,E1 34724.396,E2 34724.396} C_VEL
LIN {X 0,Y 736.075,Z 405.54,A -85,B 0,C 180,E1 34721.712,E2 34721.712} C_VEL
LIN {X 0,Y 736.013,Z 405.543,A -85,B 0,C 180,E1 34718.816,E2 34718.816} C_VEL
LIN {X 0,Y 735.998,Z 405.543,A -85,B 0,C 180,E1 34716.495,E2 34716.495} C_VEL
LIN {X 0,Y 735.997,Z 405.543,A -85,B 0,C 180,E1 34714.231,E2 34714.231} C_VEL
LIN {X 0,Y 736.042,Z 405.543,A -85,B 0,C 180,E1 34711.678,E2 34711.678} C_VEL
LIN {X 0,Y 736.007,Z 405.543,A -85,B 0,C 180,E1 34708.707,E2 34708.707} C_VEL
LIN {X 0,Y 735.987,Z 405.545,A -85,B 0,C 180,E1 34706.337,E2 34706.337} C_VEL
LIN {X 0,Y 735.99,Z 405.538,A -85,B 0,C 180,E1 34704.062,E2 34704.062} C_VEL
LIN {X 0,Y 736.028,Z 405.544,A -85,B 0,C 180,E1 34701.615,E2 34701.615} C_VEL
LIN {X 0,Y 736.018,Z 405.54,A -85,B 0,C 180,E1 34698.578,E2 34698.578} C_VEL
LIN {X 0,Y 735.998,Z 405.544,A -85,B 0,C 180,E1 34696.143,E2 34696.143} C_VEL
LIN {X 0,Y 736.005,Z 405.539,A -85,B 0,C 180,E1 34693.831,E2 34693.831} C_VEL
LIN {X 0,Y 736.098,Z 405.535,A -85,B 0,C 180,E1 34691.071,E2 34691.071} C_VEL
LIN {X 0,Y 736.018,Z 405.541,A -85,B 0,C 180,E1 34688.259,E2 34688.259} C_VEL
LIN {X 0,Y 736.061,Z 405.801,A -85,B 0,C 180,E1 34686.271,E2 34686.271} C_VEL
LIN {X 0,Y 738.722,Z 413.57,A -85,B 0,C 180,E1 34685.562,E2 34685.562} C_VEL
LIN {X 0,Y 738.309,Z 454.138,A -85,B 0,C 180,E1 34682.847,E2 34682.847} C_VEL
LIN {X 0,Y 737.922,Z 494.461,A -85,B 0,C 180,E1 34680.224,E2 34680.224} C_VEL
LIN {X 0,Y 738.003,Z 499.413,A -85,B 0,C 180,E1 34679.933,E2 34679.933} C_VEL
LIN {X 0,Y 738.933,Z 504.824,A -85,B 0,C 180,E1 34679.828,E2 34679.828} C_VEL
LIN {X 0,Y 738.415,Z 768.377,A -85,B 0,C 180,E1 34676.994,E2 34676.994} C_VEL
LIN {X 0,Y 738.239,Z 847.018,A -85,B 0,C 180,E1 34676.139,E2 34676.139} C_VEL
LIN {X 0,Y 738.106,Z 870.414,A -85,B 0,C 180,E1 34675.74,E2 34675.74} C_VEL
LIN {X 0,Y 737.974,Z 891.896,A -85,B 0,C 180,E1 34675.246,E2 34675.246} C_VEL
LIN {X 0,Y 737.735,Z 914.074,A -85,B 0,C 180,E1 34674.588,E2 34674.588} C_VEL
LIN {X 0,Y 737.577,Z 935.193,A -85,B 0,C 180,E1 34673.827,E2 34673.827} C_VEL
LIN {X 0,Y 737.317,Z 956.348,A -85,B 0,C 180,E1 34672.905,E2 34672.905} C_VEL
LIN {X 0,Y 737.098,Z 976.77,A -85,B 0,C 180,E1 34671.866,E2 34671.866} C_VEL
LIN {X 0,Y 736.882,Z 995.676,A -85,B 0,C 180,E1 34670.742,E2 34670.742} C_VEL
LIN {X 0,Y 736.645,Z 1014.898,A -85,B 0,C 180,E1 34669.424,E2 34669.424} C_VEL
LIN {X 0,Y 736.493,Z 1031.601,A -85,B 0,C 180,E1 34668.114,E2 34668.114} C_VEL
LIN {X 0,Y 736.331,Z 1047.708,A -85,B 0,C 180,E1 34666.65,E2 34666.65} C_VEL
LIN {X 0,Y 736.173,Z 1063.138,A -85,B 0,C 180,E1 34665.036,E2 34665.036} C_VEL
LIN {X 0,Y 736.09,Z 1075.776,A -85,B 0,C 180,E1 34663.512,E2 34663.512} C_VEL
LIN {X 0,Y 736.016,Z 1087.038,A -85,B 0,C 180,E1 34661.917,E2 34661.917} C_VEL
LIN {X 0,Y 735.983,Z 1097.142,A -85,B 0,C 180,E1 34660.252,E2 34660.252} C_VEL
LIN {X 0,Y 735.925,Z 1105.344,A -85,B 0,C 180,E1 34658.595,E2 34658.595} C_VEL
LIN {X 0,Y 735.911,Z 1112.393,A -85,B 0,C 180,E1 34656.867,E2 34656.867} C_VEL
LIN {X 0,Y 735.915,Z 1117.842,A -85,B 0,C 180,E1 34655.067,E2 34655.067} C_VEL
LIN {X 0,Y 735.898,Z 1121.717,A -85,B 0,C 180,E1 34653.271,E2 34653.271} C_VEL
LIN {X 0,Y 735.89,Z 1123.785,A -85,B 0,C 180,E1 34651.557,E2 34651.557} C_VEL
LIN {X 0,Y 735.902,Z 1124.452,A -85,B 0,C 180,E1 34649.766,E2 34649.766} C_VEL
LIN {X 0,Y 735.909,Z 1123.529,A -85,B 0,C 180,E1 34648.053,E2 34648.053} C_VEL
LIN {X 0,Y 735.898,Z 1120.865,A -85,B 0,C 180,E1 34646.183,E2 34646.183} C_VEL
LIN {X 0,Y 735.903,Z 1117.051,A -85,B 0,C 180,E1 34644.542,E2 34644.542} C_VEL
LIN {X 0,Y 735.926,Z 1110.927,A -85,B 0,C 180,E1 34642.662,E2 34642.662} C_VEL
LIN {X 0,Y 735.927,Z 1104.331,A -85,B 0,C 180,E1 34641.09,E2 34641.09} C_VEL
LIN {X 0,Y 735.969,Z 1094.904,A -85,B 0,C 180,E1 34639.273,E2 34639.273} C_VEL
LIN {X 0,Y 736.042,Z 1085.031,A -85,B 0,C 180,E1 34637.685,E2 34637.685} C_VEL
LIN {X 0,Y 736.115,Z 1073.301,A -85,B 0,C 180,E1 34636.088,E2 34636.088} C_VEL
LIN {X 0,Y 736.215,Z 1060.395,A -85,B 0,C 180,E1 34634.562,E2 34634.562} C_VEL
LIN {X 0,Y 736.332,Z 1046.099,A -85,B 0,C 180,E1 34633.106,E2 34633.106} C_VEL
LIN {X 0,Y 736.502,Z 1030.202,A -85,B 0,C 180,E1 34631.682,E2 34631.682} C_VEL
LIN {X 0,Y 736.663,Z 1013.584,A -85,B 0,C 180,E1 34630.388,E2 34630.388} C_VEL
LIN {X 0,Y 736.887,Z 994.464,A -85,B 0,C 180,E1 34629.092,E2 34629.092} C_VEL
LIN {X 0,Y 737.125,Z 975.482,A -85,B 0,C 180,E1 34627.972,E2 34627.972} C_VEL
LIN {X 0,Y 737.328,Z 954.686,A -85,B 0,C 180,E1 34626.926,E2 34626.926} C_VEL
LIN {X 0,Y 737.588,Z 933.091,A -85,B 0,C 180,E1 34626.003,E2 34626.003} C_VEL
LIN {X 0,Y 737.743,Z 912.942,A -85,B 0,C 180,E1 34625.284,E2 34625.284} C_VEL
LIN {X 0,Y 737.98,Z 888.935,A -85,B 0,C 180,E1 34624.591,E2 34624.591} C_VEL
LIN {X 0,Y 738.111,Z 868.138,A -85,B 0,C 180,E1 34624.123,E2 34624.123} C_VEL
LIN {X 0,Y 738.245,Z 844.278,A -85,B 0,C 180,E1 34623.737,E2 34623.737} C_VEL
LIN {X 0,Y 738.742,Z 587.599,A -85,B 0,C 180,E1 34620.979,E2 34620.979} C_VEL
LIN {X 0,Y 738.728,Z 502.724,A -85,B 0,C 180,E1 34620.05,E2 34620.05} C_VEL
LIN {X 0,Y 737.912,Z 498.676,A -85,B 0,C 180,E1 34619.95,E2 34619.95} C_VEL
LIN {X 0,Y 738.278,Z 458.973,A -85,B 0,C 180,E1 34617.382,E2 34617.382} C_VEL
LIN {X 0,Y 738.684,Z 417.218,A -85,B 0,C 180,E1 34614.595,E2 34614.595} C_VEL
LIN {X 0,Y 738.503,Z 412.591,A -85,B 0,C 180,E1 34614.268,E2 34614.268} C_VEL
LIN {X 0,Y 736.063,Z 405.721,A -85,B 0,C 180,E1 34613.624,E2 34613.624} C_VEL
LIN {X 0,Y 736.078,Z 405.544,A -85,B 0,C 180,E1 34610.741,E2 34610.741} C_VEL
LIN {X 0,Y 736.013,Z 405.544,A -85,B 0,C 180,E1 34608.057,E2 34608.057} C_VEL
LIN {X 0,Y 736.018,Z 405.536,A -85,B 0,C 180,E1 34605.609,E2 34605.609} C_VEL
LIN {X 0,Y 736.084,Z 405.541,A -85,B 0,C 180,E1 34602.702,E2 34602.702} C_VEL
LIN {X 0,Y 736.004,Z 405.543,A -85,B 0,C 180,E1 34599.984,E2 34599.984} C_VEL
LIN {X 0,Y 735.999,Z 405.543,A -85,B 0,C 180,E1 34597.687,E2 34597.687} C_VEL
LIN {X 0,Y 736.021,Z 405.536,A -85,B 0,C 180,E1 34595.266,E2 34595.266} C_VEL
LIN {X 0,Y 736.02,Z 405.543,A -85,B 0,C 180,E1 34592.177,E2 34592.177} C_VEL
LIN {X 0,Y 735.99,Z 405.545,A -85,B 0,C 180,E1 34589.758,E2 34589.758} C_VEL
LIN {X 0,Y 735.986,Z 405.544,A -85,B 0,C 180,E1 34587.511,E2 34587.511} C_VEL
LIN {X 0,Y 736.025,Z 405.545,A -85,B 0,C 180,E1 34584.992,E2 34584.992} C_VEL
LIN {X 0,Y 736.019,Z 405.543,A -85,B 0,C 180,E1 34582.021,E2 34582.021} C_VEL
LIN {X 0,Y 735.996,Z 405.543,A -85,B 0,C 180,E1 34579.607,E2 34579.607} C_VEL
LIN {X 0,Y 735.999,Z 405.543,A -85,B 0,C 180,E1 34577.309,E2 34577.309} C_VEL
LIN {X 0,Y 736.042,Z 405.544,A -85,B 0,C 180,E1 34574.797,E2 34574.797} C_VEL
LIN {X 0,Y 736.033,Z 405.54,A -85,B 0,C 180,E1 34571.837,E2 34571.837} C_VEL
LIN {X 0,Y 736.008,Z 405.541,A -85,B 0,C 180,E1 34569.383,E2 34569.383} C_VEL
LIN {X 0,Y 736.018,Z 405.541,A -85,B 0,C 180,E1 34567.023,E2 34567.023} C_VEL
LIN {X 0,Y 736.103,Z 405.538,A -85,B 0,C 180,E1 34564.207,E2 34564.207} C_VEL
LIN {X 0,Y 736.023,Z 405.54,A -85,B 0,C 180,E1 34561.401,E2 34561.401} C_VEL
LIN {X 0,Y 736.026,Z 405.539,A -85,B 0,C 180,E1 34558.91,E2 34558.91} C_VEL
LIN {X 0,Y 736.099,Z 405.537,A -85,B 0,C 180,E1 34556.028,E2 34556.028} C_VEL
LIN {X 0,Y 736.03,Z 405.539,A -85,B 0,C 180,E1 34553.212,E2 34553.212} C_VEL
LIN {X 0,Y 736.039,Z 405.541,A -85,B 0,C 180,E1 34550.697,E2 34550.697} C_VEL
LIN {X 0,Y 736.098,Z 405.535,A -85,B 0,C 180,E1 34547.766,E2 34547.766} C_VEL
LIN {X 0,Y 736.036,Z 405.537,A -85,B 0,C 180,E1 34544.991,E2 34544.991} C_VEL
LIN {X 0,Y 736.075,Z 405.543,A -85,B 0,C 180,E1 34542.285,E2 34542.285} C_VEL
LIN {X 0,Y 736.062,Z 405.535,A -85,B 0,C 180,E1 34539.234,E2 34539.234} C_VEL
LIN {X 0,Y 736.049,Z 405.54,A -85,B 0,C 180,E1 34536.545,E2 34536.545} C_VEL
LIN {X 0,Y 736.094,Z 405.538,A -85,B 0,C 180,E1 34533.706,E2 34533.706} C_VEL
LIN {X 0,Y 736.054,Z 405.535,A -85,B 0,C 180,E1 34530.866,E2 34530.866} C_VEL
LIN {X 0,Y 736.083,Z 405.544,A -85,B 0,C 180,E1 34528.101,E2 34528.101} C_VEL
LIN {X 0,Y 736.078,Z 405.531,A -85,B 0,C 180,E1 34525.023,E2 34525.023} C_VEL
LIN {X 0,Y 736.076,Z 405.543,A -85,B 0,C 180,E1 34522.12,E2 34522.12} C_VEL
LIN {X 0,Y 736.092,Z 405.533,A -85,B 0,C 180,E1 34519.1,E2 34519.1} C_VEL
LIN {X 0,Y 736.065,Z 405.537,A -85,B 0,C 180,E1 34516.256,E2 34516.256} C_VEL
LIN {X 0,Y 736.084,Z 405.535,A -85,B 0,C 180,E1 34513.386,E2 34513.386} C_VEL
LIN {X 0,Y 736.075,Z 405.538,A -85,B 0,C 180,E1 34510.593,E2 34510.593} C_VEL
LIN {X 0,Y 736.094,Z 405.534,A -85,B 0,C 180,E1 34507.681,E2 34507.681} C_VEL
LIN {X 0,Y 736.119,Z 405.757,A -85,B 0,C 180,E1 34507.039,E2 34507.039} C_VEL
LIN {X 0,Y 738.953,Z 413.432,A -85,B 0,C 180,E1 34506.347,E2 34506.347} C_VEL
LIN {X 0,Y 738.651,Z 452.804,A -85,B 0,C 180,E1 34503.882,E2 34503.882} C_VEL
LIN {X 0,Y 739.782,Z 458.73,A -85,B 0,C 180,E1 34503.751,E2 34503.751} C_VEL
LIN {X 0,Y 739.147,Z 714.906,A -85,B 0,C 180,E1 34500.897,E2 34500.897} C_VEL
LIN {X 0,Y 738.87,Z 842.622,A -85,B 0,C 180,E1 34499.481,E2 34499.481} C_VEL
LIN {X 0,Y 738.664,Z 867.847,A -85,B 0,C 180,E1 34499.064,E2 34499.064} C_VEL
LIN {X 0,Y 738.509,Z 889.354,A -85,B 0,C 180,E1 34498.576,E2 34498.576} C_VEL
LIN {X 0,Y 738.318,Z 912.614,A -85,B 0,C 180,E1 34497.92,E2 34497.92} C_VEL
LIN {X 0,Y 738.045,Z 935.538,A -85,B 0,C 180,E1 34497.115,E2 34497.115} C_VEL
LIN {X 0,Y 737.827,Z 956.229,A -85,B 0,C 180,E1 34496.262,E2 34496.262} C_VEL
LIN {X 0,Y 737.505,Z 979.137,A -85,B 0,C 180,E1 34495.153,E2 34495.153} C_VEL
LIN {X 0,Y 737.28,Z 998.883,A -85,B 0,C 180,E1 34494.05,E2 34494.05} C_VEL
LIN {X 0,Y 736.993,Z 1019.232,A -85,B 0,C 180,E1 34492.747,E2 34492.747} C_VEL
LIN {X 0,Y 736.789,Z 1037.104,A -85,B 0,C 180,E1 34491.449,E2 34491.449} C_VEL
LIN {X 0,Y 736.563,Z 1054.602,A -85,B 0,C 180,E1 34490.005,E2 34490.005} C_VEL
LIN {X 0,Y 736.424,Z 1070.493,A -85,B 0,C 180,E1 34488.525,E2 34488.525} C_VEL
LIN {X 0,Y 736.241,Z 1085.801,A -85,B 0,C 180,E1 34486.896,E2 34486.896} C_VEL
LIN {X 0,Y 736.14,Z 1098.715,A -85,B 0,C 180,E1 34485.336,E2 34485.336} C_VEL
LIN {X 0,Y 736.044,Z 1111.753,A -85,B 0,C 180,E1 34483.512,E2 34483.512} C_VEL
LIN {X 0,Y 735.992,Z 1121.12,A -85,B 0,C 180,E1 34481.994,E2 34481.994} C_VEL
LIN {X 0,Y 735.959,Z 1130.76,A -85,B 0,C 180,E1 34480.173,E2 34480.173} C_VEL
LIN {X 0,Y 735.92,Z 1138.206,A -85,B 0,C 180,E1 34478.438,E2 34478.438} C_VEL
LIN {X 0,Y 735.917,Z 1143.997,A -85,B 0,C 180,E1 34476.789,E2 34476.789} C_VEL
LIN {X 0,Y 735.898,Z 1149.178,A -85,B 0,C 180,E1 34474.832,E2 34474.832} C_VEL
LIN {X 0,Y 735.892,Z 1152.122,A -85,B 0,C 180,E1 34473.194,E2 34473.194} C_VEL
LIN {X 0,Y 735.905,Z 1154.099,A -85,B 0,C 180,E1 34471.324,E2 34471.324} C_VEL
LIN {X 0,Y 735.881,Z 1154.351,A -85,B 0,C 180,E1 34469.455,E2 34469.455} C_VEL
LIN {X 0,Y 735.917,Z 1153.297,A -85,B 0,C 180,E1 34467.742,E2 34467.742} C_VEL
LIN {X 0,Y 735.915,Z 1150.288,A -85,B 0,C 180,E1 34465.714,E2 34465.714} C_VEL
LIN {X 0,Y 735.923,Z 1146.353,A -85,B 0,C 180,E1 34464.024,E2 34464.024} C_VEL
LIN {X 0,Y 735.915,Z 1140.271,A -85,B 0,C 180,E1 34462.096,E2 34462.096} C_VEL
LIN {X 0,Y 735.932,Z 1133.245,A -85,B 0,C 180,E1 34460.38,E2 34460.38} C_VEL
LIN {X 0,Y 735.965,Z 1125.11,A -85,B 0,C 180,E1 34458.718,E2 34458.718} C_VEL
LIN {X 0,Y 736.02,Z 1114.352,A -85,B 0,C 180,E1 34456.887,E2 34456.887} C_VEL
LIN {X 0,Y 736.109,Z 1103.953,A -85,B 0,C 180,E1 34455.365,E2 34455.365} C_VEL
LIN {X 0,Y 736.227,Z 1090.044,A -85,B 0,C 180,E1 34453.591,E2 34453.591} C_VEL
LIN {X 0,Y 736.329,Z 1076.067,A -85,B 0,C 180,E1 34452.046,E2 34452.046} C_VEL
LIN {X 0,Y 736.53,Z 1059.246,A -85,B 0,C 180,E1 34450.408,E2 34450.408} C_VEL
LIN {X 0,Y 736.711,Z 1042.805,A -85,B 0,C 180,E1 34449.003,E2 34449.003} C_VEL
LIN {X 0,Y 736.963,Z 1022.853,A -85,B 0,C 180,E1 34447.504,E2 34447.504} C_VEL
LIN {X 0,Y 737.195,Z 1004.357,A -85,B 0,C 180,E1 34446.282,E2 34446.282} C_VEL
LIN {X 0,Y 737.48,Z 982.344,A -85,B 0,C 180,E1 34445.018,E2 34445.018} C_VEL
LIN {X 0,Y 737.72,Z 962.785,A -85,B 0,C 180,E1 34444.037,E2 34444.037} C_VEL
LIN {X 0,Y 738.022,Z 939.382,A -85,B 0,C 180,E1 34443.034,E2 34443.034} C_VEL
LIN {X 0,Y 738.199,Z 919.691,A -85,B 0,C 180,E1 34442.316,E2 34442.316} C_VEL
LIN {X 0,Y 738.492,Z 896.035,A -85,B 0,C 180,E1 34441.595,E2 34441.595} C_VEL
LIN {X 0,Y 738.638,Z 873.308,A -85,B 0,C 180,E1 34441.051,E2 34441.051} C_VEL
LIN {X 0,Y 738.792,Z 852.207,A -85,B 0,C 180,E1 34440.658,E2 34440.658} C_VEL
LIN {X 0,Y 738.923,Z 821.026,A -85,B 0,C 180,E1 34440.263,E2 34440.263} C_VEL
LIN {X 0,Y 739.426,Z 581.429,A -85,B 0,C 180,E1 34437.624,E2 34437.624} C_VEL
LIN {X 0,Y 739.609,Z 456.974,A -85,B 0,C 180,E1 34436.22,E2 34436.22} C_VEL
LIN {X 0,Y 738.576,Z 452.077,A -85,B 0,C 180,E1 34436.087,E2 34436.087} C_VEL
LIN {X 0,Y 738.952,Z 413.432,A -85,B 0,C 180,E1 34433.653,E2 34433.653} C_VEL
LIN {X 0,Y 736.117,Z 405.748,A -85,B 0,C 180,E1 34432.961,E2 34432.961} C_VEL
LIN {X 0,Y 736.089,Z 405.541,A -85,B 0,C 180,E1 34430.122,E2 34430.122} C_VEL
LIN {X 0,Y 736.089,Z 405.529,A -85,B 0,C 180,E1 34427.113,E2 34427.113} C_VEL
LIN {X 0,Y 736.089,Z 405.537,A -85,B 0,C 180,E1 34424.062,E2 34424.062} C_VEL
LIN {X 0,Y 736.08,Z 405.534,A -85,B 0,C 180,E1 34421.107,E2 34421.107} C_VEL
LIN {X 0,Y 736.092,Z 405.54,A -85,B 0,C 180,E1 34418.076,E2 34418.076} C_VEL
LIN {X 0,Y 736.058,Z 405.534,A -85,B 0,C 180,E1 34415.264,E2 34415.264} C_VEL
LIN {X 0,Y 736.091,Z 405.532,A -85,B 0,C 180,E1 34412.45,E2 34412.45} C_VEL
LIN {X 0,Y 736.06,Z 405.539,A -85,B 0,C 180,E1 34409.611,E2 34409.611} C_VEL
LIN {X 0,Y 736.074,Z 405.534,A -85,B 0,C 180,E1 34406.807,E2 34406.807} C_VEL
LIN {X 0,Y 736.07,Z 405.542,A -85,B 0,C 180,E1 34403.709,E2 34403.709} C_VEL
LIN {X 0,Y 736.046,Z 405.537,A -85,B 0,C 180,E1 34401.016,E2 34401.016} C_VEL
LIN {X 0,Y 736.097,Z 405.536,A -85,B 0,C 180,E1 34398.206,E2 34398.206} C_VEL
LIN {X 0,Y 736.047,Z 405.54,A -85,B 0,C 180,E1 34395.361,E2 34395.361} C_VEL
LIN {X 0,Y 736.047,Z 405.537,A -85,B 0,C 180,E1 34392.713,E2 34392.713} C_VEL
LIN {X 0,Y 736.097,Z 405.541,A -85,B 0,C 180,E1 34389.776,E2 34389.776} C_VEL
LIN {X 0,Y 736.03,Z 405.54,A -85,B 0,C 180,E1 34387.023,E2 34387.023} C_VEL
LIN {X 0,Y 736.052,Z 405.536,A -85,B 0,C 180,E1 34384.441,E2 34384.441} C_VEL
LIN {X 0,Y 736.05,Z 405.54,A -85,B 0,C 180,E1 34381.323,E2 34381.323} C_VEL
LIN {X 0,Y 736.023,Z 405.541,A -85,B 0,C 180,E1 34378.832,E2 34378.832} C_VEL
LIN {X 0,Y 736.047,Z 405.536,A -85,B 0,C 180,E1 34376.261,E2 34376.261} C_VEL
LIN {X 0,Y 736.045,Z 405.542,A -85,B 0,C 180,E1 34373.213,E2 34373.213} C_VEL
LIN {X 0,Y 736.013,Z 405.541,A -85,B 0,C 180,E1 34370.696,E2 34370.696} C_VEL
LIN {X 0,Y 736.047,Z 405.543,A -85,B 0,C 180,E1 34369.189,E2 34369.189} C_VEL
LIN {X 0,Y 735.003,Z 405.669,A -85,B 0,C 180,E1 34368.589,E2 34368.589} C_VEL
LIN {X 0,Y 728.59,Z 406.469,A -85,B 0,C 180,E1 34366.909,E2 34366.909} C_VEL
LIN {X 0,Y 728.071,Z 406.53,A -85,B 0,C 180,E1 34366.473,E2 34366.473} C_VEL
LIN {X 0,Y 728.115,Z 406.53,A -85,B 0,C 180,E1 34363.895,E2 34363.895} C_VEL
LIN {X 0,Y 728.08,Z 406.532,A -85,B 0,C 180,E1 34360.883,E2 34360.883} C_VEL
LIN {X 0,Y 728.06,Z 406.531,A -85,B 0,C 180,E1 34358.488,E2 34358.488} C_VEL
LIN {X 0,Y 728.066,Z 406.532,A -85,B 0,C 180,E1 34356.157,E2 34356.157} C_VEL
LIN {X 0,Y 728.154,Z 406.533,A -85,B 0,C 180,E1 34353.318,E2 34353.318} C_VEL
LIN {X 0,Y 728.057,Z 406.534,A -85,B 0,C 180,E1 34350.55,E2 34350.55} C_VEL
LIN {X 0,Y 728.048,Z 406.532,A -85,B 0,C 180,E1 34348.226,E2 34348.226} C_VEL
LIN {X 0,Y 728.067,Z 406.534,A -85,B 0,C 180,E1 34345.826,E2 34345.826} C_VEL
LIN {X 0,Y 728.092,Z 406.533,A -85,B 0,C 180,E1 34342.799,E2 34342.799} C_VEL
LIN {X 0,Y 728.054,Z 406.532,A -85,B 0,C 180,E1 34340.273,E2 34340.273} C_VEL
LIN {X 0,Y 728.058,Z 406.529,A -85,B 0,C 180,E1 34337.987,E2 34337.987} C_VEL
LIN {X 0,Y 728.123,Z 406.534,A -85,B 0,C 180,E1 34335.323,E2 34335.323} C_VEL
LIN {X 0,Y 728.077,Z 406.533,A -85,B 0,C 180,E1 34332.366,E2 34332.366} C_VEL
LIN {X 0,Y 728.066,Z 406.531,A -85,B 0,C 180,E1 34329.974,E2 34329.974} C_VEL
LIN {X 0,Y 728.083,Z 406.529,A -85,B 0,C 180,E1 34327.572,E2 34327.572} C_VEL
LIN {X 0,Y 728.174,Z 406.822,A -85,B 0,C 180,E1 34326.654,E2 34326.654} C_VEL
LIN {X 0,Y 731.667,Z 416.841,A -85,B 0,C 180,E1 34325.732,E2 34325.732} C_VEL
LIN {X 0,Y 731.12,Z 457.623,A -85,B 0,C 180,E1 34322.978,E2 34322.978} C_VEL
LIN {X 0,Y 730.617,Z 497.251,A -85,B 0,C 180,E1 34320.377,E2 34320.377} C_VEL
LIN {X 0,Y 730.821,Z 499.96,A -85,B 0,C 180,E1 34320.249,E2 34320.249} C_VEL
LIN {X 0,Y 731.988,Z 506.376,A -85,B 0,C 180,E1 34320.123,E2 34320.123} C_VEL
LIN {X 0,Y 731.282,Z 769.711,A -85,B 0,C 180,E1 34317.266,E2 34317.266} C_VEL
LIN {X 0,Y 731.051,Z 847.169,A -85,B 0,C 180,E1 34316.414,E2 34316.414} C_VEL
LIN {X 0,Y 730.868,Z 870.427,A -85,B 0,C 180,E1 34316.014,E2 34316.014} C_VEL
LIN {X 0,Y 730.689,Z 892.352,A -85,B 0,C 180,E1 34315.505,E2 34315.505} C_VEL
LIN {X 0,Y 730.377,Z 914.094,A -85,B 0,C 180,E1 34314.853,E2 34314.853} C_VEL
LIN {X 0,Y 730.158,Z 935.21,A -85,B 0,C 180,E1 34314.085,E2 34314.085} C_VEL
LIN {X 0,Y 729.811,Z 956.363,A -85,B 0,C 180,E1 34313.154,E2 34313.154} C_VEL
LIN {X 0,Y 729.504,Z 977.584,A -85,B 0,C 180,E1 34312.059,E2 34312.059} C_VEL
LIN {X 0,Y 729.217,Z 996.347,A -85,B 0,C 180,E1 34310.928,E2 34310.928} C_VEL
LIN {X 0,Y 728.915,Z 1014.906,A -85,B 0,C 180,E1 34309.638,E2 34309.638} C_VEL
LIN {X 0,Y 728.693,Z 1032.017,A -85,B 0,C 180,E1 34308.278,E2 34308.278} C_VEL
LIN {X 0,Y 728.475,Z 1047.714,A -85,B 0,C 180,E1 34306.835,E2 34306.835} C_VEL
LIN {X 0,Y 728.274,Z 1063.144,A -85,B 0,C 180,E1 34305.203,E2 34305.203} C_VEL
LIN {X 0,Y 728.161,Z 1075.778,A -85,B 0,C 180,E1 34303.662,E2 34303.662} C_VEL
LIN {X 0,Y 728.063,Z 1087.042,A -85,B 0,C 180,E1 34302.049,E2 34302.049} C_VEL
LIN {X 0,Y 728.004,Z 1097.144,A -85,B 0,C 180,E1 34300.365,E2 34300.365} C_VEL
LIN {X 0,Y 727.936,Z 1105.346,A -85,B 0,C 180,E1 34298.69,E2 34298.69} C_VEL
LIN {X 0,Y 727.92,Z 1112.395,A -85,B 0,C 180,E1 34296.943,E2 34296.943} C_VEL
LIN {X 0,Y 727.917,Z 1117.843,A -85,B 0,C 180,E1 34295.123,E2 34295.123} C_VEL
LIN {X 0,Y 727.896,Z 1121.717,A -85,B 0,C 180,E1 34293.307,E2 34293.307} C_VEL
LIN {X 0,Y 727.891,Z 1123.785,A -85,B 0,C 180,E1 34291.574,E2 34291.574} C_VEL
LIN {X 0,Y 727.902,Z 1124.452,A -85,B 0,C 180,E1 34289.764,E2 34289.764} C_VEL
LIN {X 0,Y 727.909,Z 1123.529,A -85,B 0,C 180,E1 34288.032,E2 34288.032} C_VEL
LIN {X 0,Y 727.901,Z 1120.865,A -85,B 0,C 180,E1 34286.141,E2 34286.141} C_VEL
LIN {X 0,Y 727.902,Z 1117.05,A -85,B 0,C 180,E1 34284.482,E2 34284.482} C_VEL
LIN {X 0,Y 727.926,Z 1110.925,A -85,B 0,C 180,E1 34282.581,E2 34282.581} C_VEL
LIN {X 0,Y 727.945,Z 1104.24,A -85,B 0,C 180,E1 34280.971,E2 34280.971} C_VEL
LIN {X 0,Y 727.995,Z 1094.902,A -85,B 0,C 180,E1 34279.154,E2 34279.154} C_VEL
LIN {X 0,Y 728.088,Z 1084.942,A -85,B 0,C 180,E1 34277.535,E2 34277.535} C_VEL
LIN {X 0,Y 728.189,Z 1072.657,A -85,B 0,C 180,E1 34275.853,E2 34275.853} C_VEL
LIN {X 0,Y 728.346,Z 1059.668,A -85,B 0,C 180,E1 34274.309,E2 34274.309} C_VEL
LIN {X 0,Y 728.506,Z 1044.868,A -85,B 0,C 180,E1 34272.8,E2 34272.8} C_VEL
LIN {X 0,Y 728.741,Z 1027.665,A -85,B 0,C 180,E1 34271.272,E2 34271.272} C_VEL
LIN {X 0,Y 729.025,Z 1009.975,A -85,B 0,C 180,E1 34269.905,E2 34269.905} C_VEL
LIN {X 0,Y 729.288,Z 991.152,A -85,B 0,C 180,E1 34268.653,E2 34268.653} C_VEL
LIN {X 0,Y 729.601,Z 970.619,A -85,B 0,C 180,E1 34267.473,E2 34267.473} C_VEL
LIN {X 0,Y 729.909,Z 951.087,A -85,B 0,C 180,E1 34266.507,E2 34266.507} C_VEL
LIN {X 0,Y 730.191,Z 929.117,A -85,B 0,C 180,E1 34265.592,E2 34265.592} C_VEL
LIN {X 0,Y 730.521,Z 907.068,A -85,B 0,C 180,E1 34264.828,E2 34264.828} C_VEL
LIN {X 0,Y 730.721,Z 884.773,A -85,B 0,C 180,E1 34264.215,E2 34264.215} C_VEL
LIN {X 0,Y 730.964,Z 861.037,A -85,B 0,C 180,E1 34263.716,E2 34263.716} C_VEL
LIN {X 0,Y 731.071,Z 839.973,A -85,B 0,C 180,E1 34263.404,E2 34263.404} C_VEL
LIN {X 0,Y 731.737,Z 588.791,A -85,B 0,C 180,E1 34260.688,E2 34260.688} C_VEL
LIN {X 0,Y 731.791,Z 504.277,A -85,B 0,C 180,E1 34259.754,E2 34259.754} C_VEL
LIN {X 0,Y 730.622,Z 498.447,A -85,B 0,C 180,E1 34259.606,E2 34259.606} C_VEL
LIN {X 0,Y 731.109,Z 458.964,A -85,B 0,C 180,E1 34257.022,E2 34257.022} C_VEL
LIN {X 0,Y 731.649,Z 418.183,A -85,B 0,C 180,E1 34254.27,E2 34254.27} C_VEL
LIN {X 0,Y 731.443,Z 415.816,A -85,B 0,C 180,E1 34254.094,E2 34254.094} C_VEL
LIN {X 0,Y 728.177,Z 406.718,A -85,B 0,C 180,E1 34253.237,E2 34253.237} C_VEL
LIN {X 0,Y 728.087,Z 406.531,A -85,B 0,C 180,E1 34250.313,E2 34250.313} C_VEL
LIN {X 0,Y 728.073,Z 406.533,A -85,B 0,C 180,E1 34247.868,E2 34247.868} C_VEL
LIN {X 0,Y 728.123,Z 406.522,A -85,B 0,C 180,E1 34245.213,E2 34245.213} C_VEL
LIN {X 0,Y 728.082,Z 406.528,A -85,B 0,C 180,E1 34242.249,E2 34242.249} C_VEL
LIN {X 0,Y 728.062,Z 406.531,A -85,B 0,C 180,E1 34239.851,E2 34239.851} C_VEL
LIN {X 0,Y 728.065,Z 406.532,A -85,B 0,C 180,E1 34237.573,E2 34237.573} C_VEL
LIN {X 0,Y 728.159,Z 406.524,A -85,B 0,C 180,E1 34234.741,E2 34234.741} C_VEL
LIN {X 0,Y 728.059,Z 406.532,A -85,B 0,C 180,E1 34231.921,E2 34231.921} C_VEL
LIN {X 0,Y 728.05,Z 406.534,A -85,B 0,C 180,E1 34229.616,E2 34229.616} C_VEL
LIN {X 0,Y 728.057,Z 406.533,A -85,B 0,C 180,E1 34227.304,E2 34227.304} C_VEL
LIN {X 0,Y 728.134,Z 406.533,A -85,B 0,C 180,E1 34224.415,E2 34224.415} C_VEL
LIN {X 0,Y 728.059,Z 406.532,A -85,B 0,C 180,E1 34221.766,E2 34221.766} C_VEL
LIN {X 0,Y 728.057,Z 406.533,A -85,B 0,C 180,E1 34219.412,E2 34219.412} C_VEL
LIN {X 0,Y 728.089,Z 406.532,A -85,B 0,C 180,E1 34216.926,E2 34216.926} C_VEL
LIN {X 0,Y 728.086,Z 406.53,A -85,B 0,C 180,E1 34213.825,E2 34213.825} C_VEL
LIN {X 0,Y 728.067,Z 406.53,A -85,B 0,C 180,E1 34211.406,E2 34211.406} C_VEL
LIN {X 0,Y 728.079,Z 406.531,A -85,B 0,C 180,E1 34209.007,E2 34209.007} C_VEL
LIN {X 0,Y 728.159,Z 406.528,A -85,B 0,C 180,E1 34206.149,E2 34206.149} C_VEL
LIN {X 0,Y 728.079,Z 406.527,A -85,B 0,C 180,E1 34203.385,E2 34203.385} C_VEL
LIN {X 0,Y 728.085,Z 406.531,A -85,B 0,C 180,E1 34200.944,E2 34200.944} C_VEL
LIN {X 0,Y 728.162,Z 406.529,A -85,B 0,C 180,E1 34198.111,E2 34198.111} C_VEL
LIN {X 0,Y 728.089,Z 406.527,A -85,B 0,C 180,E1 34195.274,E2 34195.274} C_VEL
LIN {X 0,Y 728.097,Z 406.53,A -85,B 0,C 180,E1 34192.742,E2 34192.742} C_VEL
LIN {X 0,Y 728.158,Z 406.524,A -85,B 0,C 180,E1 34189.797,E2 34189.797} C_VEL
LIN {X 0,Y 728.096,Z 406.528,A -85,B 0,C 180,E1 34187.065,E2 34187.065} C_VEL
LIN {X 0,Y 728.117,Z 406.53,A -85,B 0,C 180,E1 34184.467,E2 34184.467} C_VEL
LIN {X 0,Y 728.138,Z 406.522,A -85,B 0,C 180,E1 34181.422,E2 34181.422} C_VEL
LIN {X 0,Y 728.105,Z 406.529,A -85,B 0,C 180,E1 34178.659,E2 34178.659} C_VEL
LIN {X 0,Y 728.155,Z 406.529,A -85,B 0,C 180,E1 34175.845,E2 34175.845} C_VEL
LIN {X 0,Y 728.116,Z 406.525,A -85,B 0,C 180,E1 34172.964,E2 34172.964} C_VEL
LIN {X 0,Y 728.136,Z 406.53,A -85,B 0,C 180,E1 34170.191,E2 34170.191} C_VEL
LIN {X 0,Y 728.137,Z 406.517,A -85,B 0,C 180,E1 34167.058,E2 34167.058} C_VEL
LIN {X 0,Y 728.131,Z 406.528,A -85,B 0,C 180,E1 34164.197,E2 34164.197} C_VEL
LIN {X 0,Y 728.157,Z 406.514,A -85,B 0,C 180,E1 34161.232,E2 34161.232} C_VEL
LIN {X 0,Y 728.121,Z 406.528,A -85,B 0,C 180,E1 34158.449,E2 34158.449} C_VEL
LIN {X 0,Y 728.152,Z 406.525,A -85,B 0,C 180,E1 34155.657,E2 34155.657} C_VEL
LIN {X 0,Y 728.14,Z 406.519,A -85,B 0,C 180,E1 34152.716,E2 34152.716} C_VEL
LIN {X 0,Y 728.159,Z 406.525,A -85,B 0,C 180,E1 34149.737,E2 34149.737} C_VEL
LIN {X 0,Y 728.18,Z 406.771,A -85,B 0,C 180,E1 34147.442,E2 34147.442} C_VEL
LIN {X 0,Y 731.996,Z 417.159,A -85,B 0,C 180,E1 34146.505,E2 34146.505} C_VEL
LIN {X 0,Y 731.602,Z 452.844,A -85,B 0,C 180,E1 34144.253,E2 34144.253} C_VEL
LIN {X 0,Y 733.118,Z 460.422,A -85,B 0,C 180,E1 34144.08,E2 34144.08} C_VEL
LIN {X 0,Y 732.273,Z 716.051,A -85,B 0,C 180,E1 34141.207,E2 34141.207} C_VEL
LIN {X 0,Y 731.896,Z 842.73,A -85,B 0,C 180,E1 34139.788,E2 34139.788} C_VEL
LIN {X 0,Y 731.63,Z 868.109,A -85,B 0,C 180,E1 34139.365,E2 34139.365} C_VEL
LIN {X 0,Y 731.416,Z 889.68,A -85,B 0,C 180,E1 34138.87,E2 34138.87} C_VEL
LIN {X 0,Y 731.15,Z 913.285,A -85,B 0,C 180,E1 34138.196,E2 34138.196} C_VEL
LIN {X 0,Y 730.784,Z 936.272,A -85,B 0,C 180,E1 34137.378,E2 34137.378} C_VEL
LIN {X 0,Y 730.481,Z 958.075,A -85,B 0,C 180,E1 34136.465,E2 34136.465} C_VEL
LIN {X 0,Y 730.06,Z 979.943,A -85,B 0,C 180,E1 34135.384,E2 34135.384} C_VEL
LIN {X 0,Y 729.749,Z 1000.341,A -85,B 0,C 180,E1 34134.228,E2 34134.228} C_VEL
LIN {X 0,Y 729.366,Z 1020.441,A -85,B 0,C 180,E1 34132.913,E2 34132.913} C_VEL
LIN {X 0,Y 729.084,Z 1039.25,A -85,B 0,C 180,E1 34131.522,E2 34131.522} C_VEL
LIN {X 0,Y 728.776,Z 1056.46,A -85,B 0,C 180,E1 34130.06,E2 34130.06} C_VEL
LIN {X 0,Y 728.567,Z 1072.961,A -85,B 0,C 180,E1 34128.483,E2 34128.483} C_VEL
LIN {X 0,Y 728.355,Z 1087.454,A -85,B 0,C 180,E1 34126.893,E2 34126.893} C_VEL
LIN {X 0,Y 728.207,Z 1101.057,A -85,B 0,C 180,E1 34125.204,E2 34125.204} C_VEL
LIN {X 0,Y 728.086,Z 1112.793,A -85,B 0,C 180,E1 34123.501,E2 34123.501} C_VEL
LIN {X 0,Y 728.02,Z 1122.95,A -85,B 0,C 180,E1 34121.809,E2 34121.809} C_VEL
LIN {X 0,Y 727.95,Z 1132.181,A -85,B 0,C 180,E1 34119.966,E2 34119.966} C_VEL
LIN {X 0,Y 727.932,Z 1138.815,A -85,B 0,C 180,E1 34118.372,E2 34118.372} C_VEL
LIN {X 0,Y 727.912,Z 1145.245,A -85,B 0,C 180,E1 34116.467,E2 34116.467} C_VEL
LIN {X 0,Y 727.917,Z 1149.813,A -85,B 0,C 180,E1 34114.57,E2 34114.57} C_VEL
LIN {X 0,Y 727.882,Z 1152.684,A -85,B 0,C 180,E1 34112.835,E2 34112.835} C_VEL
LIN {X 0,Y 727.89,Z 1154.262,A -85,B 0,C 180,E1 34110.866,E2 34110.866} C_VEL
LIN {X 0,Y 727.883,Z 1154.306,A -85,B 0,C 180,E1 34109.292,E2 34109.292} C_VEL
LIN {X 0,Y 727.89,Z 1153.017,A -85,B 0,C 180,E1 34107.402,E2 34107.402} C_VEL
LIN {X 0,Y 727.916,Z 1149.971,A -85,B 0,C 180,E1 34105.509,E2 34105.509} C_VEL
LIN {X 0,Y 727.92,Z 1145.864,A -85,B 0,C 180,E1 34103.77,E2 34103.77} C_VEL
LIN {X 0,Y 727.942,Z 1139.422,A -85,B 0,C 180,E1 34101.787,E2 34101.787} C_VEL
LIN {X 0,Y 727.944,Z 1132.891,A -85,B 0,C 180,E1 34100.193,E2 34100.193} C_VEL
LIN {X 0,Y 728.023,Z 1124.295,A -85,B 0,C 180,E1 34098.433,E2 34098.433} C_VEL
LIN {X 0,Y 728.073,Z 1113.834,A -85,B 0,C 180,E1 34096.66,E2 34096.66} C_VEL
LIN {X 0,Y 728.18,Z 1103.376,A -85,B 0,C 180,E1 34095.121,E2 34095.121} C_VEL
LIN {X 0,Y 728.355,Z 1088.632,A -85,B 0,C 180,E1 34093.244,E2 34093.244} C_VEL
LIN {X 0,Y 728.507,Z 1075.291,A -85,B 0,C 180,E1 34091.764,E2 34091.764} C_VEL
LIN {X 0,Y 728.757,Z 1058.318,A -85,B 0,C 180,E1 34090.107,E2 34090.107} C_VEL
LIN {X 0,Y 729.027,Z 1041.791,A -85,B 0,C 180,E1 34088.687,E2 34088.687} C_VEL
LIN {X 0,Y 729.343,Z 1022.251,A -85,B 0,C 180,E1 34087.214,E2 34087.214} C_VEL
LIN {X 0,Y 729.684,Z 1003.76,A -85,B 0,C 180,E1 34085.985,E2 34085.985} C_VEL
LIN {X 0,Y 730.032,Z 982.347,A -85,B 0,C 180,E1 34084.745,E2 34084.745} C_VEL
LIN {X 0,Y 730.389,Z 962.155,A -85,B 0,C 180,E1 34083.726,E2 34083.726} C_VEL
LIN {X 0,Y 730.764,Z 938.712,A -85,B 0,C 180,E1 34082.718,E2 34082.718} C_VEL
LIN {X 0,Y 731.018,Z 918.422,A -85,B 0,C 180,E1 34081.976,E2 34081.976} C_VEL
LIN {X 0,Y 731.401,Z 892.947,A -85,B 0,C 180,E1 34081.214,E2 34081.214} C_VEL
LIN {X 0,Y 731.604,Z 871.754,A -85,B 0,C 180,E1 34080.712,E2 34080.712} C_VEL
LIN {X 0,Y 731.874,Z 847.924,A -85,B 0,C 180,E1 34080.28,E2 34080.28} C_VEL
LIN {X 0,Y 732.008,Z 806.775,A -85,B 0,C 180,E1 34079.795,E2 34079.795} C_VEL
LIN {X 0,Y 732.685,Z 573.616,A -85,B 0,C 180,E1 34077.2,E2 34077.2} C_VEL
LIN {X 0,Y 732.957,Z 458.719,A -85,B 0,C 180,E1 34075.892,E2 34075.892} C_VEL
LIN {X 0,Y 731.525,Z 452.274,A -85,B 0,C 180,E1 34075.726,E2 34075.726} C_VEL
LIN {X 0,Y 731.9,Z 416.502,A -85,B 0,C 180,E1 34073.447,E2 34073.447} C_VEL
LIN {X 0,Y 728.178,Z 406.766,A -85,B 0,C 180,E1 34072.558,E2 34072.558} C_VEL
LIN {X 0,Y 728.135,Z 406.533,A -85,B 0,C 180,E1 34069.897,E2 34069.897} C_VEL
LIN {X 0,Y 728.155,Z 406.518,A -85,B 0,C 180,E1 34066.963,E2 34066.963} C_VEL
LIN {X 0,Y 728.142,Z 406.524,A -85,B 0,C 180,E1 34063.981,E2 34063.981} C_VEL
LIN {X 0,Y 728.148,Z 406.522,A -85,B 0,C 180,E1 34061.025,E2 34061.025} C_VEL
LIN {X 0,Y 728.147,Z 406.531,A -85,B 0,C 180,E1 34057.966,E2 34057.966} C_VEL
LIN {X 0,Y 728.131,Z 406.521,A -85,B 0,C 180,E1 34055.07,E2 34055.07} C_VEL
LIN {X 0,Y 728.154,Z 406.528,A -85,B 0,C 180,E1 34052.085,E2 34052.085} C_VEL
LIN {X 0,Y 728.112,Z 406.525,A -85,B 0,C 180,E1 34049.267,E2 34049.267} C_VEL
LIN {X 0,Y 728.157,Z 406.524,A -85,B 0,C 180,E1 34046.451,E2 34046.451} C_VEL
LIN {X 0,Y 728.118,Z 406.53,A -85,B 0,C 180,E1 34043.554,E2 34043.554} C_VEL
LIN {X 0,Y 728.118,Z 406.525,A -85,B 0,C 180,E1 34040.835,E2 34040.835} C_VEL
LIN {X 0,Y 728.153,Z 406.531,A -85,B 0,C 180,E1 34037.832,E2 34037.832} C_VEL
LIN {X 0,Y 728.099,Z 406.526,A -85,B 0,C 180,E1 34035.044,E2 34035.044} C_VEL
LIN {X 0,Y 728.157,Z 406.523,A -85,B 0,C 180,E1 34032.289,E2 34032.289} C_VEL
LIN {X 0,Y 728.107,Z 406.53,A -85,B 0,C 180,E1 34029.326,E2 34029.326} C_VEL
LIN {X 0,Y 728.097,Z 406.527,A -85,B 0,C 180,E1 34026.703,E2 34026.703} C_VEL
LIN {X 0,Y 728.159,Z 406.53,A -85,B 0,C 180,E1 34023.779,E2 34023.779} C_VEL
LIN {X 0,Y 728.088,Z 406.527,A -85,B 0,C 180,E1 34021.023,E2 34021.023} C_VEL
LIN {X 0,Y 728.093,Z 406.528,A -85,B 0,C 180,E1 34018.505,E2 34018.505} C_VEL
LIN {X 0,Y 728.156,Z 406.53,A -85,B 0,C 180,E1 34015.59,E2 34015.59} C_VEL
LIN {X 0,Y 728.081,Z 406.529,A -85,B 0,C 180,E1 34012.9,E2 34012.9} C_VEL
LIN {X 0,Y 728.077,Z 406.529,A -85,B 0,C 180,E1 34010.514,E2 34010.514} C_VEL
LIN {X 0,Y 728.147,Z 406.528,A -85,B 0,C 180,E1 34007.791,E2 34007.791} C_VEL
LIN {X 0,Y 728.071,Z 406.53,A -85,B 0,C 180,E1 34006.473,E2 34006.473} C_VEL
LIN {X 0,Y 727.083,Z 406.659,A -85,B 0,C 180,E1 34005.867,E2 34005.867} C_VEL
LIN {X 0,Y 720.776,Z 407.442,A -85,B 0,C 180,E1 34004.212,E2 34004.212} C_VEL
LIN {X 0,Y 720.202,Z 407.518,A -85,B 0,C 180,E1 34003.728,E2 34003.728} C_VEL
LIN {X 0,Y 720.135,Z 407.521,A -85,B 0,C 180,E1 34000.788,E2 34000.788} C_VEL
LIN {X 0,Y 720.121,Z 407.52,A -85,B 0,C 180,E1 33998.41,E2 33998.41} C_VEL
LIN {X 0,Y 720.14,Z 407.52,A -85,B 0,C 180,E1 33995.995,E2 33995.995} C_VEL
LIN {X 0,Y 720.149,Z 407.521,A -85,B 0,C 180,E1 33992.908,E2 33992.908} C_VEL
LIN {X 0,Y 720.114,Z 407.523,A -85,B 0,C 180,E1 33990.467,E2 33990.467} C_VEL
LIN {X 0,Y 720.111,Z 407.521,A -85,B 0,C 180,E1 33988.154,E2 33988.154} C_VEL
LIN {X 0,Y 720.161,Z 407.523,A -85,B 0,C 180,E1 33985.561,E2 33985.561} C_VEL
LIN {X 0,Y 720.13,Z 407.522,A -85,B 0,C 180,E1 33982.582,E2 33982.582} C_VEL
LIN {X 0,Y 720.114,Z 407.521,A -85,B 0,C 180,E1 33980.2,E2 33980.2} C_VEL
LIN {X 0,Y 720.125,Z 407.517,A -85,B 0,C 180,E1 33977.856,E2 33977.856} C_VEL
LIN {X 0,Y 720.21,Z 407.509,A -85,B 0,C 180,E1 33974.964,E2 33974.964} C_VEL
LIN {X 0,Y 720.13,Z 407.523,A -85,B 0,C 180,E1 33972.224,E2 33972.224} C_VEL
LIN {X 0,Y 720.13,Z 407.52,A -85,B 0,C 180,E1 33969.84,E2 33969.84} C_VEL
LIN {X 0,Y 720.202,Z 407.552,A -85,B 0,C 180,E1 33967.152,E2 33967.152} C_VEL
LIN {X 0,Y 720.394,Z 408.457,A -85,B 0,C 180,E1 33966.986,E2 33966.986} C_VEL
LIN {X 0,Y 724.619,Z 420.111,A -85,B 0,C 180,E1 33965.904,E2 33965.904} C_VEL
LIN {X 0,Y 723.934,Z 461.109,A -85,B 0,C 180,E1 33963.111,E2 33963.111} C_VEL
LIN {X 0,Y 723.39,Z 498.967,A -85,B 0,C 180,E1 33960.614,E2 33960.614} C_VEL
LIN {X 0,Y 725.063,Z 507.822,A -85,B 0,C 180,E1 33960.426,E2 33960.426} C_VEL
LIN {X 0,Y 724.166,Z 771.285,A -85,B 0,C 180,E1 33957.539,E2 33957.539} C_VEL
LIN {X 0,Y 723.881,Z 847.319,A -85,B 0,C 180,E1 33956.695,E2 33956.695} C_VEL
LIN {X 0,Y 723.647,Z 870.594,A -85,B 0,C 180,E1 33956.291,E2 33956.291} C_VEL
LIN {X 0,Y 723.418,Z 892.915,A -85,B 0,C 180,E1 33955.766,E2 33955.766} C_VEL
LIN {X 0,Y 723.03,Z 914.812,A -85,B 0,C 180,E1 33955.099,E2 33955.099} C_VEL
LIN {X 0,Y 722.73,Z 936.26,A -85,B 0,C 180,E1 33954.305,E2 33954.305} C_VEL
LIN {X 0,Y 722.308,Z 957.268,A -85,B 0,C 180,E1 33953.366,E2 33953.366} C_VEL
LIN {X 0,Y 721.92,Z 978.325,A -85,B 0,C 180,E1 33952.26,E2 33952.26} C_VEL
LIN {X 0,Y 721.561,Z 997.02,A -85,B 0,C 180,E1 33951.118,E2 33951.118} C_VEL
LIN {X 0,Y 721.194,Z 1015.262,A -85,B 0,C 180,E1 33949.831,E2 33949.831} C_VEL
LIN {X 0,Y 720.896,Z 1032.544,A -85,B 0,C 180,E1 33948.436,E2 33948.436} C_VEL
LIN {X 0,Y 720.629,Z 1047.72,A -85,B 0,C 180,E1 33947.024,E2 33947.024} C_VEL
LIN {X 0,Y 720.387,Z 1063.15,A -85,B 0,C 180,E1 33945.373,E2 33945.373} C_VEL
LIN {X 0,Y 720.237,Z 1075.781,A -85,B 0,C 180,E1 33943.815,E2 33943.815} C_VEL
LIN {X 0,Y 720.108,Z 1087.143,A -85,B 0,C 180,E1 33942.169,E2 33942.169} C_VEL
LIN {X 0,Y 720.025,Z 1097.146,A -85,B 0,C 180,E1 33940.482,E2 33940.482} C_VEL
LIN {X 0,Y 719.948,Z 1105.349,A -85,B 0,C 180,E1 33938.788,E2 33938.788} C_VEL
LIN {X 0,Y 719.93,Z 1112.397,A -85,B 0,C 180,E1 33937.02,E2 33937.02} C_VEL
LIN {X 0,Y 719.917,Z 1117.845,A -85,B 0,C 180,E1 33935.18,E2 33935.18} C_VEL
LIN {X 0,Y 719.895,Z 1121.717,A -85,B 0,C 180,E1 33933.344,E2 33933.344} C_VEL
LIN {X 0,Y 719.891,Z 1123.786,A -85,B 0,C 180,E1 33931.592,E2 33931.592} C_VEL
LIN {X 0,Y 719.902,Z 1124.451,A -85,B 0,C 180,E1 33929.761,E2 33929.761} C_VEL
LIN {X 0,Y 719.91,Z 1123.529,A -85,B 0,C 180,E1 33928.01,E2 33928.01} C_VEL
LIN {X 0,Y 719.904,Z 1120.865,A -85,B 0,C 180,E1 33926.098,E2 33926.098} C_VEL
LIN {X 0,Y 719.902,Z 1117.049,A -85,B 0,C 180,E1 33924.421,E2 33924.421} C_VEL
LIN {X 0,Y 719.928,Z 1110.923,A -85,B 0,C 180,E1 33922.498,E2 33922.498} C_VEL
LIN {X 0,Y 719.963,Z 1104.328,A -85,B 0,C 180,E1 33920.89,E2 33920.89} C_VEL
LIN {X 0,Y 720.025,Z 1094.9,A -85,B 0,C 180,E1 33919.033,E2 33919.033} C_VEL
LIN {X 0,Y 720.134,Z 1085.027,A -85,B 0,C 180,E1 33917.409,E2 33917.409} C_VEL
LIN {X 0,Y 720.267,Z 1072.647,A -85,B 0,C 180,E1 33915.693,E2 33915.693} C_VEL
LIN {X 0,Y 720.463,Z 1059.435,A -85,B 0,C 180,E1 33914.108,E2 33914.108} C_VEL
LIN {X 0,Y 720.67,Z 1045.239,A -85,B 0,C 180,E1 33912.644,E2 33912.644} C_VEL
LIN {X 0,Y 720.962,Z 1028.165,A -85,B 0,C 180,E1 33911.105,E2 33911.105} C_VEL
LIN {X 0,Y 721.314,Z 1010.546,A -85,B 0,C 180,E1 33909.723,E2 33909.723} C_VEL
LIN {X 0,Y 721.653,Z 991.807,A -85,B 0,C 180,E1 33908.459,E2 33908.459} C_VEL
LIN {X 0,Y 722.05,Z 970.787,A -85,B 0,C 180,E1 33907.233,E2 33907.233} C_VEL
LIN {X 0,Y 722.449,Z 951.071,A -85,B 0,C 180,E1 33906.25,E2 33906.25} C_VEL
LIN {X 0,Y 722.792,Z 929.765,A -85,B 0,C 180,E1 33905.351,E2 33905.351} C_VEL
LIN {X 0,Y 723.203,Z 907.757,A -85,B 0,C 180,E1 33904.577,E2 33904.577} C_VEL
LIN {X 0,Y 723.461,Z 885.34,A -85,B 0,C 180,E1 33903.952,E2 33903.952} C_VEL
LIN {X 0,Y 723.764,Z 862.141,A -85,B 0,C 180,E1 33903.454,E2 33903.454} C_VEL
LIN {X 0,Y 723.905,Z 840.573,A -85,B 0,C 180,E1 33903.128,E2 33903.128} C_VEL
LIN {X 0,Y 724.747,Z 590.289,A -85,B 0,C 180,E1 33900.394,E2 33900.394} C_VEL
LIN {X 0,Y 724.857,Z 505.778,A -85,B 0,C 180,E1 33899.452,E2 33899.452} C_VEL
LIN {X 0,Y 723.369,Z 498.527,A -85,B 0,C 180,E1 33899.273,E2 33899.273} C_VEL
LIN {X 0,Y 723.993,Z 457.562,A -85,B 0,C 180,E1 33896.561,E2 33896.561} C_VEL
LIN {X 0,Y 724.604,Z 419.766,A -85,B 0,C 180,E1 33893.98,E2 33893.98} C_VEL
LIN {X 0,Y 720.238,Z 407.707,A -85,B 0,C 180,E1 33892.833,E2 33892.833} C_VEL
LIN {X 0,Y 720.141,Z 407.52,A -85,B 0,C 180,E1 33890.159,E2 33890.159} C_VEL
LIN {X 0,Y 720.139,Z 407.522,A -85,B 0,C 180,E1 33887.736,E2 33887.736} C_VEL
LIN {X 0,Y 720.219,Z 407.51,A -85,B 0,C 180,E1 33884.851,E2 33884.851} C_VEL
LIN {X 0,Y 720.133,Z 407.516,A -85,B 0,C 180,E1 33882.116,E2 33882.116} C_VEL
LIN {X 0,Y 720.124,Z 407.52,A -85,B 0,C 180,E1 33879.715,E2 33879.715} C_VEL
LIN {X 0,Y 720.151,Z 407.52,A -85,B 0,C 180,E1 33877.255,E2 33877.255} C_VEL
LIN {X 0,Y 720.139,Z 407.522,A -85,B 0,C 180,E1 33874.154,E2 33874.154} C_VEL
LIN {X 0,Y 720.114,Z 407.52,A -85,B 0,C 180,E1 33871.752,E2 33871.752} C_VEL
LIN {X 0,Y 720.116,Z 407.523,A -85,B 0,C 180,E1 33869.442,E2 33869.442} C_VEL
LIN {X 0,Y 720.205,Z 407.522,A -85,B 0,C 180,E1 33866.643,E2 33866.643} C_VEL
LIN {X 0,Y 720.121,Z 407.522,A -85,B 0,C 180,E1 33863.832,E2 33863.832} C_VEL
LIN {X 0,Y 720.114,Z 407.521,A -85,B 0,C 180,E1 33861.504,E2 33861.504} C_VEL
LIN {X 0,Y 720.131,Z 407.522,A -85,B 0,C 180,E1 33859.128,E2 33859.128} C_VEL
LIN {X 0,Y 720.191,Z 407.52,A -85,B 0,C 180,E1 33856.204,E2 33856.204} C_VEL
LIN {X 0,Y 720.13,Z 407.519,A -85,B 0,C 180,E1 33853.571,E2 33853.571} C_VEL
LIN {X 0,Y 720.13,Z 407.52,A -85,B 0,C 180,E1 33851.209,E2 33851.209} C_VEL
LIN {X 0,Y 720.208,Z 407.519,A -85,B 0,C 180,E1 33848.463,E2 33848.463} C_VEL
LIN {X 0,Y 720.148,Z 407.518,A -85,B 0,C 180,E1 33845.578,E2 33845.578} C_VEL
LIN {X 0,Y 720.139,Z 407.516,A -85,B 0,C 180,E1 33843.104,E2 33843.104} C_VEL
LIN {X 0,Y 720.218,Z 407.519,A -85,B 0,C 180,E1 33840.318,E2 33840.318} C_VEL
LIN {X 0,Y 720.153,Z 407.518,A -85,B 0,C 180,E1 33837.374,E2 33837.374} C_VEL
LIN {X 0,Y 720.153,Z 407.518,A -85,B 0,C 180,E1 33834.822,E2 33834.822} C_VEL
LIN {X 0,Y 720.222,Z 407.515,A -85,B 0,C 180,E1 33831.939,E2 33831.939} C_VEL
LIN {X 0,Y 720.156,Z 407.516,A -85,B 0,C 180,E1 33829.116,E2 33829.116} C_VEL
LIN {X 0,Y 720.185,Z 407.52,A -85,B 0,C 180,E1 33826.43,E2 33826.43} C_VEL
LIN {X 0,Y 720.183,Z 407.514,A -85,B 0,C 180,E1 33823.333,E2 33823.333} C_VEL
LIN {X 0,Y 720.167,Z 407.517,A -85,B 0,C 180,E1 33820.62,E2 33820.62} C_VEL
LIN {X 0,Y 720.218,Z 407.514,A -85,B 0,C 180,E1 33817.727,E2 33817.727} C_VEL
LIN {X 0,Y 720.17,Z 407.515,A -85,B 0,C 180,E1 33814.857,E2 33814.857} C_VEL
LIN {X 0,Y 720.22,Z 407.521,A -85,B 0,C 180,E1 33812.003,E2 33812.003} C_VEL
LIN {X 0,Y 720.189,Z 407.514,A -85,B 0,C 180,E1 33808.997,E2 33808.997} C_VEL
LIN {X 0,Y 720.199,Z 407.51,A -85,B 0,C 180,E1 33806.123,E2 33806.123} C_VEL
LIN {X 0,Y 720.208,Z 407.512,A -85,B 0,C 180,E1 33803.048,E2 33803.048} C_VEL
LIN {X 0,Y 720.195,Z 407.509,A -85,B 0,C 180,E1 33800.102,E2 33800.102} C_VEL
LIN {X 0,Y 720.215,Z 407.506,A -85,B 0,C 180,E1 33797.025,E2 33797.025} C_VEL
LIN {X 0,Y 720.198,Z 407.521,A -85,B 0,C 180,E1 33794.073,E2 33794.073} C_VEL
LIN {X 0,Y 720.216,Z 407.516,A -85,B 0,C 180,E1 33791.047,E2 33791.047} C_VEL
LIN {X 0,Y 720.194,Z 407.525,A -85,B 0,C 180,E1 33788.157,E2 33788.157} C_VEL
LIN {X 0,Y 720.276,Z 407.938,A -85,B 0,C 180,E1 33787.831,E2 33787.831} C_VEL
LIN {X 0,Y 725.036,Z 420.42,A -85,B 0,C 180,E1 33786.697,E2 33786.697} C_VEL
LIN {X 0,Y 724.591,Z 452.918,A -85,B 0,C 180,E1 33784.63,E2 33784.63} C_VEL
LIN {X 0,Y 726.479,Z 462.091,A -85,B 0,C 180,E1 33784.415,E2 33784.415} C_VEL
LIN {X 0,Y 725.421,Z 717.451,A -85,B 0,C 180,E1 33781.519,E2 33781.519} C_VEL
LIN {X 0,Y 724.941,Z 842.837,A -85,B 0,C 180,E1 33780.102,E2 33780.102} C_VEL
LIN {X 0,Y 724.618,Z 868.368,A -85,B 0,C 180,E1 33779.672,E2 33779.672} C_VEL
LIN {X 0,Y 724.342,Z 890.115,A -85,B 0,C 180,E1 33779.168,E2 33779.168} C_VEL
LIN {X 0,Y 724.014,Z 913.281,A -85,B 0,C 180,E1 33778.499,E2 33778.499} C_VEL
LIN {X 0,Y 723.568,Z 935.358,A -85,B 0,C 180,E1 33777.711,E2 33777.711} C_VEL
LIN {X 0,Y 723.176,Z 957.231,A -85,B 0,C 180,E1 33776.791,E2 33776.791} C_VEL
LIN {X 0,Y 722.68,Z 979.144,A -85,B 0,C 180,E1 33775.706,E2 33775.706} C_VEL
LIN {X 0,Y 722.248,Z 999.617,A -85,B 0,C 180,E1 33774.54,E2 33774.54} C_VEL
LIN {X 0,Y 721.8,Z 1019.839,A -85,B 0,C 180,E1 33773.211,E2 33773.211} C_VEL
LIN {X 0,Y 721.413,Z 1038.708,A -85,B 0,C 180,E1 33771.805,E2 33771.805} C_VEL
LIN {X 0,Y 721.03,Z 1056.46,A -85,B 0,C 180,E1 33770.285,E2 33770.285} C_VEL
LIN {X 0,Y 720.756,Z 1072.963,A -85,B 0,C 180,E1 33768.691,E2 33768.691} C_VEL
LIN {X 0,Y 720.478,Z 1087.219,A -85,B 0,C 180,E1 33767.111,E2 33767.111} C_VEL
LIN {X 0,Y 720.295,Z 1101.059,A -85,B 0,C 180,E1 33765.375,E2 33765.375} C_VEL
LIN {X 0,Y 720.142,Z 1113.081,A -85,B 0,C 180,E1 33763.608,E2 33763.608} C_VEL
LIN {X 0,Y 720.049,Z 1123.867,A -85,B 0,C 180,E1 33761.779,E2 33761.779} C_VEL
LIN {X 0,Y 719.96,Z 1132.892,A -85,B 0,C 180,E1 33759.917,E2 33759.917} C_VEL
LIN {X 0,Y 719.944,Z 1139.423,A -85,B 0,C 180,E1 33758.305,E2 33758.305} C_VEL
LIN {X 0,Y 719.92,Z 1146.07,A -85,B 0,C 180,E1 33756.219,E2 33756.219} C_VEL
LIN {X 0,Y 719.917,Z 1149.972,A -85,B 0,C 180,E1 33754.541,E2 33754.541} C_VEL
LIN {X 0,Y 719.888,Z 1153.017,A -85,B 0,C 180,E1 33752.627,E2 33752.627} C_VEL
LIN {X 0,Y 719.883,Z 1154.306,A -85,B 0,C 180,E1 33750.716,E2 33750.716} C_VEL
LIN {X 0,Y 719.896,Z 1154.24,A -85,B 0,C 180,E1 33749.045,E2 33749.045} C_VEL
LIN {X 0,Y 719.882,Z 1152.559,A -85,B 0,C 180,E1 33747.045,E2 33747.045} C_VEL
LIN {X 0,Y 719.916,Z 1149.813,A -85,B 0,C 180,E1 33745.379,E2 33745.379} C_VEL
LIN {X 0,Y 719.916,Z 1145.245,A -85,B 0,C 180,E1 33743.46,E2 33743.46} C_VEL
LIN {X 0,Y 719.934,Z 1138.814,A -85,B 0,C 180,E1 33741.534,E2 33741.534} C_VEL
LIN {X 0,Y 719.973,Z 1132.181,A -85,B 0,C 180,E1 33739.922,E2 33739.922} C_VEL
LIN {X 0,Y 720.055,Z 1122.031,A -85,B 0,C 180,E1 33737.896,E2 33737.896} C_VEL
LIN {X 0,Y 720.156,Z 1112.276,A -85,B 0,C 180,E1 33736.265,E2 33736.265} C_VEL
LIN {X 0,Y 720.315,Z 1099.681,A -85,B 0,C 180,E1 33734.444,E2 33734.444} C_VEL
LIN {X 0,Y 720.49,Z 1086.512,A -85,B 0,C 180,E1 33732.806,E2 33732.806} C_VEL
LIN {X 0,Y 720.782,Z 1071.334,A -85,B 0,C 180,E1 33731.142,E2 33731.142} C_VEL
LIN {X 0,Y 721.057,Z 1055.43,A -85,B 0,C 180,E1 33729.622,E2 33729.622} C_VEL
LIN {X 0,Y 721.426,Z 1037.603,A -85,B 0,C 180,E1 33728.11,E2 33728.11} C_VEL
LIN {X 0,Y 721.817,Z 1019.235,A -85,B 0,C 180,E1 33726.747,E2 33726.747} C_VEL
LIN {X 0,Y 722.275,Z 997.433,A -85,B 0,C 180,E1 33725.33,E2 33725.33} C_VEL
LIN {X 0,Y 722.725,Z 977.524,A -85,B 0,C 180,E1 33724.208,E2 33724.208} C_VEL
LIN {X 0,Y 723.206,Z 954.252,A -85,B 0,C 180,E1 33723.077,E2 33723.077} C_VEL
LIN {X 0,Y 723.625,Z 933.105,A -85,B 0,C 180,E1 33722.202,E2 33722.202} C_VEL
LIN {X 0,Y 724.069,Z 908.958,A -85,B 0,C 180,E1 33721.368,E2 33721.368} C_VEL
LIN {X 0,Y 724.364,Z 887.095,A -85,B 0,C 180,E1 33720.754,E2 33720.754} C_VEL
LIN {X 0,Y 724.745,Z 862.436,A -85,B 0,C 180,E1 33720.212,E2 33720.212} C_VEL
LIN {X 0,Y 724.951,Z 839.812,A -85,B 0,C 180,E1 33719.858,E2 33719.858} C_VEL
LIN {X 0,Y 725.916,Z 584.483,A -85,B 0,C 180,E1 33716.981,E2 33716.981} C_VEL
LIN {X 0,Y 726.29,Z 460.289,A -85,B 0,C 180,E1 33715.553,E2 33715.553} C_VEL
LIN {X 0,Y 724.498,Z 452.169,A -85,B 0,C 180,E1 33715.341,E2 33715.341} C_VEL
LIN {X 0,Y 724.903,Z 419.953,A -85,B 0,C 180,E1 33713.264,E2 33713.264} C_VEL
LIN {X 0,Y 720.253,Z 407.812,A -85,B 0,C 180,E1 33712.149,E2 33712.149} C_VEL
LIN {X 0,Y 720.203,Z 407.511,A -85,B 0,C 180,E1 33710.722,E2 33710.722} C_VEL
LIN {X 0,Y 720.193,Z 407.509,A -85,B 0,C 180,E1 33707.85,E2 33707.85} C_VEL
LIN {X 0,Y 720.217,Z 407.512,A -85,B 0,C 180,E1 33704.924,E2 33704.924} C_VEL
LIN {X 0,Y 720.199,Z 407.521,A -85,B 0,C 180,E1 33701.898,E2 33701.898} C_VEL
LIN {X 0,Y 720.209,Z 407.501,A -85,B 0,C 180,E1 33698.97,E2 33698.97} C_VEL
LIN {X 0,Y 720.2,Z 407.517,A -85,B 0,C 180,E1 33695.866,E2 33695.866} C_VEL
LIN {X 0,Y 720.196,Z 407.506,A -85,B 0,C 180,E1 33692.973,E2 33692.973} C_VEL
LIN {X 0,Y 720.209,Z 407.518,A -85,B 0,C 180,E1 33689.895,E2 33689.895} C_VEL
LIN {X 0,Y 720.176,Z 407.515,A -85,B 0,C 180,E1 33687.09,E2 33687.09} C_VEL
LIN {X 0,Y 720.218,Z 407.517,A -85,B 0,C 180,E1 33684.177,E2 33684.177} C_VEL
LIN {X 0,Y 720.168,Z 407.518,A -85,B 0,C 180,E1 33681.332,E2 33681.332} C_VEL
LIN {X 0,Y 720.207,Z 407.51,A -85,B 0,C 180,E1 33678.515,E2 33678.515} C_VEL
LIN {X 0,Y 720.176,Z 407.518,A -85,B 0,C 180,E1 33675.46,E2 33675.46} C_VEL
LIN {X 0,Y 720.167,Z 407.515,A -85,B 0,C 180,E1 33672.754,E2 33672.754} C_VEL
LIN {X 0,Y 720.221,Z 407.517,A -85,B 0,C 180,E1 33669.832,E2 33669.832} C_VEL
LIN {X 0,Y 720.153,Z 407.518,A -85,B 0,C 180,E1 33667.018,E2 33667.018} C_VEL
LIN {X 0,Y 720.182,Z 407.513,A -85,B 0,C 180,E1 33664.379,E2 33664.379} C_VEL
LIN {X 0,Y 720.168,Z 407.517,A -85,B 0,C 180,E1 33661.273,E2 33661.273} C_VEL
LIN {X 0,Y 720.145,Z 407.519,A -85,B 0,C 180,E1 33658.727,E2 33658.727} C_VEL
LIN {X 0,Y 720.212,Z 407.512,A -85,B 0,C 180,E1 33655.94,E2 33655.94} C_VEL
LIN {X 0,Y 720.152,Z 407.519,A -85,B 0,C 180,E1 33653.062,E2 33653.062} C_VEL
LIN {X 0,Y 720.137,Z 407.519,A -85,B 0,C 180,E1 33650.57,E2 33650.57} C_VEL
LIN {X 0,Y 720.192,Z 407.517,A -85,B 0,C 180,E1 33647.898,E2 33647.898} C_VEL
LIN {X 0,Y 720.146,Z 407.521,A -85,B 0,C 180,E1 33644.951,E2 33644.951} C_VEL
LIN {X 0,Y 720.202,Z 407.518,A -85,B 0,C 180,E1 33643.728,E2 33643.728} C_VEL
LIN {X 0,Y 719.282,Z 407.642,A -85,B 0,C 180,E1 33643.115,E2 33643.115} C_VEL
LIN {X 0,Y 712.787,Z 408.448,A -85,B 0,C 180,E1 33641.4,E2 33641.4} C_VEL
LIN {X 0,Y 712.209,Z 408.511,A -85,B 0,C 180,E1 33640.953,E2 33640.953} C_VEL
LIN {X 0,Y 712.183,Z 408.509,A -85,B 0,C 180,E1 33638.504,E2 33638.504} C_VEL
LIN {X 0,Y 712.19,Z 408.51,A -85,B 0,C 180,E1 33636.15,E2 33636.15} C_VEL
LIN {X 0,Y 712.261,Z 408.51,A -85,B 0,C 180,E1 33633.232,E2 33633.232} C_VEL
LIN {X 0,Y 712.178,Z 408.512,A -85,B 0,C 180,E1 33630.514,E2 33630.514} C_VEL
LIN {X 0,Y 712.173,Z 408.509,A -85,B 0,C 180,E1 33628.149,E2 33628.149} C_VEL
LIN {X 0,Y 712.233,Z 408.512,A -85,B 0,C 180,E1 33625.496,E2 33625.496} C_VEL
LIN {X 0,Y 712.19,Z 408.511,A -85,B 0,C 180,E1 33622.561,E2 33622.561} C_VEL
LIN {X 0,Y 712.175,Z 408.51,A -85,B 0,C 180,E1 33620.174,E2 33620.174} C_VEL
LIN {X 0,Y 712.194,Z 408.505,A -85,B 0,C 180,E1 33617.74,E2 33617.74} C_VEL
LIN {X 0,Y 712.235,Z 408.497,A -85,B 0,C 180,E1 33614.735,E2 33614.735} C_VEL
LIN {X 0,Y 712.189,Z 408.513,A -85,B 0,C 180,E1 33612.152,E2 33612.152} C_VEL
LIN {X 0,Y 712.198,Z 408.51,A -85,B 0,C 180,E1 33609.702,E2 33609.702} C_VEL
LIN {X 0,Y 712.238,Z 408.695,A -85,B 0,C 180,E1 33607.499,E2 33607.499} C_VEL
LIN {X 0,Y 717.584,Z 423.392,A -85,B 0,C 180,E1 33606.081,E2 33606.081} C_VEL
LIN {X 0,Y 716.753,Z 464.594,A -85,B 0,C 180,E1 33603.247,E2 33603.247} C_VEL
LIN {X 0,Y 716.179,Z 499.121,A -85,B 0,C 180,E1 33600.953,E2 33600.953} C_VEL
LIN {X 0,Y 718.158,Z 509.325,A -85,B 0,C 180,E1 33600.733,E2 33600.733} C_VEL
LIN {X 0,Y 717.067,Z 772.608,A -85,B 0,C 180,E1 33597.821,E2 33597.821} C_VEL
LIN {X 0,Y 716.728,Z 847.47,A -85,B 0,C 180,E1 33596.982,E2 33596.982} C_VEL
LIN {X 0,Y 716.442,Z 870.761,A -85,B 0,C 180,E1 33596.572,E2 33596.572} C_VEL
LIN {X 0,Y 716.167,Z 892.939,A -85,B 0,C 180,E1 33596.046,E2 33596.046} C_VEL
LIN {X 0,Y 715.7,Z 915.288,A -85,B 0,C 180,E1 33595.358,E2 33595.358} C_VEL
LIN {X 0,Y 715.308,Z 937.273,A -85,B 0,C 180,E1 33594.53,E2 33594.53} C_VEL
LIN {X 0,Y 714.833,Z 957.33,A -85,B 0,C 180,E1 33593.623,E2 33593.623} C_VEL
LIN {X 0,Y 714.345,Z 979.065,A -85,B 0,C 180,E1 33592.466,E2 33592.466} C_VEL
LIN {X 0,Y 713.904,Z 998.353,A -85,B 0,C 180,E1 33591.27,E2 33591.27} C_VEL
LIN {X 0,Y 713.455,Z 1016.578,A -85,B 0,C 180,E1 33589.954,E2 33589.954} C_VEL
LIN {X 0,Y 713.07,Z 1034.405,A -85,B 0,C 180,E1 33588.476,E2 33588.476} C_VEL
LIN {X 0,Y 712.759,Z 1050.26,A -85,B 0,C 180,E1 33586.965,E2 33586.965} C_VEL
LIN {X 0,Y 712.472,Z 1064.568,A -85,B 0,C 180,E1 33585.382,E2 33585.382} C_VEL
LIN {X 0,Y 712.279,Z 1077.587,A -85,B 0,C 180,E1 33583.724,E2 33583.724} C_VEL
LIN {X 0,Y 712.134,Z 1088.607,A -85,B 0,C 180,E1 33582.076,E2 33582.076} C_VEL
LIN {X 0,Y 712.029,Z 1099.201,A -85,B 0,C 180,E1 33580.192,E2 33580.192} C_VEL
LIN {X 0,Y 711.96,Z 1107.121,A -85,B 0,C 180,E1 33578.48,E2 33578.48} C_VEL
LIN {X 0,Y 711.911,Z 1113.932,A -85,B 0,C 180,E1 33576.613,E2 33576.613} C_VEL
LIN {X 0,Y 711.91,Z 1118.668,A -85,B 0,C 180,E1 33574.915,E2 33574.915} C_VEL
LIN {X 0,Y 711.911,Z 1122.231,A -85,B 0,C 180,E1 33573.015,E2 33573.015} C_VEL
LIN {X 0,Y 711.898,Z 1124.12,A -85,B 0,C 180,E1 33571.207,E2 33571.207} C_VEL
LIN {X 0,Y 711.891,Z 1124.363,A -85,B 0,C 180,E1 33569.437,E2 33569.437} C_VEL
LIN {X 0,Y 711.893,Z 1123.184,A -85,B 0,C 180,E1 33567.585,E2 33567.585} C_VEL
LIN {X 0,Y 711.909,Z 1120.215,A -85,B 0,C 180,E1 33565.723,E2 33565.723} C_VEL
LIN {X 0,Y 711.929,Z 1115.734,A -85,B 0,C 180,E1 33563.873,E2 33563.873} C_VEL
LIN {X 0,Y 711.931,Z 1110.012,A -85,B 0,C 180,E1 33562.17,E2 33562.17} C_VEL
LIN {X 0,Y 711.99,Z 1102.493,A -85,B 0,C 180,E1 33560.38,E2 33560.38} C_VEL
LIN {X 0,Y 712.08,Z 1093.513,A -85,B 0,C 180,E1 33558.663,E2 33558.663} C_VEL
LIN {X 0,Y 712.219,Z 1082.259,A -85,B 0,C 180,E1 33556.854,E2 33556.854} C_VEL
LIN {X 0,Y 712.398,Z 1070.49,A -85,B 0,C 180,E1 33555.252,E2 33555.252} C_VEL
LIN {X 0,Y 712.617,Z 1056.572,A -85,B 0,C 180,E1 33553.619,E2 33553.619} C_VEL
LIN {X 0,Y 712.923,Z 1041.836,A -85,B 0,C 180,E1 33552.112,E2 33552.112} C_VEL
LIN {X 0,Y 713.26,Z 1025.628,A -85,B 0,C 180,E1 33550.68,E2 33550.68} C_VEL
LIN {X 0,Y 713.664,Z 1007.405,A -85,B 0,C 180,E1 33549.272,E2 33549.272} C_VEL
LIN {X 0,Y 714.114,Z 989.124,A -85,B 0,C 180,E1 33548.047,E2 33548.047} C_VEL
LIN {X 0,Y 714.566,Z 969.095,A -85,B 0,C 180,E1 33546.89,E2 33546.89} C_VEL
LIN {X 0,Y 715.073,Z 948.306,A -85,B 0,C 180,E1 33545.858,E2 33545.858} C_VEL
LIN {X 0,Y 715.468,Z 927.457,A -85,B 0,C 180,E1 33544.991,E2 33544.991} C_VEL
LIN {X 0,Y 715.94,Z 904.834,A -85,B 0,C 180,E1 33544.212,E2 33544.212} C_VEL
LIN {X 0,Y 716.259,Z 883.252,A -85,B 0,C 180,E1 33543.617,E2 33543.617} C_VEL
LIN {X 0,Y 716.599,Z 859.176,A -85,B 0,C 180,E1 33543.116,E2 33543.116} C_VEL
LIN {X 0,Y 716.777,Z 837.528,A -85,B 0,C 180,E1 33542.8,E2 33542.8} C_VEL
LIN {X 0,Y 717.771,Z 593.218,A -85,B 0,C 180,E1 33540.111,E2 33540.111} C_VEL
LIN {X 0,Y 717.979,Z 507.442,A -85,B 0,C 180,E1 33539.147,E2 33539.147} C_VEL
LIN {X 0,Y 716.144,Z 498.766,A -85,B 0,C 180,E1 33538.942,E2 33538.942} C_VEL
LIN {X 0,Y 716.924,Z 456.052,A -85,B 0,C 180,E1 33536.083,E2 33536.083} C_VEL
LIN {X 0,Y 717.491,Z 422.978,A -85,B 0,C 180,E1 33533.794,E2 33533.794} C_VEL
LIN {X 0,Y 712.243,Z 408.695,A -85,B 0,C 180,E1 33532.412,E2 33532.412} C_VEL
LIN {X 0,Y 712.198,Z 408.505,A -85,B 0,C 180,E1 33529.921,E2 33529.921} C_VEL
LIN {X 0,Y 712.248,Z 408.51,A -85,B 0,C 180,E1 33527.241,E2 33527.241} C_VEL
LIN {X 0,Y 712.207,Z 408.512,A -85,B 0,C 180,E1 33524.247,E2 33524.247} C_VEL
LIN {X 0,Y 712.187,Z 408.504,A -85,B 0,C 180,E1 33521.797,E2 33521.797} C_VEL
LIN {X 0,Y 712.214,Z 408.508,A -85,B 0,C 180,E1 33519.284,E2 33519.284} C_VEL
LIN {X 0,Y 712.205,Z 408.499,A -85,B 0,C 180,E1 33516.232,E2 33516.232} C_VEL
LIN {X 0,Y 712.179,Z 408.511,A -85,B 0,C 180,E1 33513.778,E2 33513.778} C_VEL
LIN {X 0,Y 712.184,Z 408.509,A -85,B 0,C 180,E1 33511.391,E2 33511.391} C_VEL
LIN {X 0,Y 712.256,Z 408.509,A -85,B 0,C 180,E1 33508.51,E2 33508.51} C_VEL
LIN {X 0,Y 712.176,Z 408.512,A -85,B 0,C 180,E1 33505.801,E2 33505.801} C_VEL
LIN {X 0,Y 712.175,Z 408.511,A -85,B 0,C 180,E1 33503.499,E2 33503.499} C_VEL
LIN {X 0,Y 712.19,Z 408.51,A -85,B 0,C 180,E1 33501.151,E2 33501.151} C_VEL
LIN {X 0,Y 712.237,Z 408.508,A -85,B 0,C 180,E1 33498.159,E2 33498.159} C_VEL
LIN {X 0,Y 712.186,Z 408.51,A -85,B 0,C 180,E1 33495.555,E2 33495.555} C_VEL
LIN {X 0,Y 712.189,Z 408.509,A -85,B 0,C 180,E1 33493.229,E2 33493.229} C_VEL
LIN {X 0,Y 712.263,Z 408.51,A -85,B 0,C 180,E1 33490.515,E2 33490.515} C_VEL
LIN {X 0,Y 712.204,Z 408.506,A -85,B 0,C 180,E1 33487.584,E2 33487.584} C_VEL
LIN {X 0,Y 712.198,Z 408.509,A -85,B 0,C 180,E1 33485.155,E2 33485.155} C_VEL
LIN {X 0,Y 712.266,Z 408.507,A -85,B 0,C 180,E1 33482.414,E2 33482.414} C_VEL
LIN {X 0,Y 712.218,Z 408.502,A -85,B 0,C 180,E1 33479.517,E2 33479.517} C_VEL
LIN {X 0,Y 712.21,Z 408.509,A -85,B 0,C 180,E1 33476.942,E2 33476.942} C_VEL
LIN {X 0,Y 712.285,Z 408.506,A -85,B 0,C 180,E1 33474.037,E2 33474.037} C_VEL
LIN {X 0,Y 712.217,Z 408.505,A -85,B 0,C 180,E1 33471.198,E2 33471.198} C_VEL
LIN {X 0,Y 712.232,Z 408.508,A -85,B 0,C 180,E1 33468.583,E2 33468.583} C_VEL
LIN {X 0,Y 712.261,Z 408.5,A -85,B 0,C 180,E1 33465.529,E2 33465.529} C_VEL
LIN {X 0,Y 712.222,Z 408.507,A -85,B 0,C 180,E1 33462.769,E2 33462.769} C_VEL
LIN {X 0,Y 712.281,Z 408.507,A -85,B 0,C 180,E1 33459.907,E2 33459.907} C_VEL
LIN {X 0,Y 712.234,Z 408.503,A -85,B 0,C 180,E1 33457.028,E2 33457.028} C_VEL
LIN {X 0,Y 712.261,Z 408.508,A -85,B 0,C 180,E1 33454.203,E2 33454.203} C_VEL
LIN {X 0,Y 712.256,Z 408.499,A -85,B 0,C 180,E1 33451.124,E2 33451.124} C_VEL
LIN {X 0,Y 712.253,Z 408.51,A -85,B 0,C 180,E1 33448.235,E2 33448.235} C_VEL
LIN {X 0,Y 712.273,Z 408.496,A -85,B 0,C 180,E1 33445.156,E2 33445.156} C_VEL
LIN {X 0,Y 712.251,Z 408.51,A -85,B 0,C 180,E1 33442.22,E2 33442.22} C_VEL
LIN {X 0,Y 712.277,Z 408.502,A -85,B 0,C 180,E1 33439.249,E2 33439.249} C_VEL
LIN {X 0,Y 712.246,Z 408.5,A -85,B 0,C 180,E1 33436.418,E2 33436.418} C_VEL
LIN {X 0,Y 712.272,Z 408.503,A -85,B 0,C 180,E1 33433.572,E2 33433.572} C_VEL
LIN {X 0,Y 712.259,Z 408.508,A -85,B 0,C 180,E1 33430.582,E2 33430.582} C_VEL
LIN {X 0,Y 712.276,Z 408.681,A -85,B 0,C 180,E1 33428.305,E2 33428.305} C_VEL
LIN {X 0,Y 714.206,Z 413.955,A -85,B 0,C 180,E1 33427.786,E2 33427.786} C_VEL
LIN {X 0,Y 718.078,Z 423.87,A -85,B 0,C 180,E1 33426.881,E2 33426.881} C_VEL
LIN {X 0,Y 717.6,Z 452.929,A -85,B 0,C 180,E1 33425.017,E2 33425.017} C_VEL
LIN {X 0,Y 719.864,Z 463.829,A -85,B 0,C 180,E1 33424.756,E2 33424.756} C_VEL
LIN {X 0,Y 718.592,Z 718.342,A -85,B 0,C 180,E1 33421.844,E2 33421.844} C_VEL
LIN {X 0,Y 718.009,Z 842.945,A -85,B 0,C 180,E1 33420.422,E2 33420.422} C_VEL
LIN {X 0,Y 717.638,Z 868.495,A -85,B 0,C 180,E1 33419.987,E2 33419.987} C_VEL
LIN {X 0,Y 717.291,Z 890.215,A -85,B 0,C 180,E1 33419.48,E2 33419.48} C_VEL
LIN {X 0,Y 716.857,Z 914.562,A -85,B 0,C 180,E1 33418.765,E2 33418.765} C_VEL
LIN {X 0,Y 716.34,Z 936.481,A -85,B 0,C 180,E1 33417.97,E2 33417.97} C_VEL
LIN {X 0,Y 715.831,Z 959.58,A -85,B 0,C 180,E1 33416.978,E2 33416.978} C_VEL
LIN {X 0,Y 715.246,Z 980.753,A -85,B 0,C 180,E1 33415.904,E2 33415.904} C_VEL
LIN {X 0,Y 714.719,Z 1001.753,A -85,B 0,C 180,E1 33414.683,E2 33414.683} C_VEL
LIN {X 0,Y 714.188,Z 1021.128,A -85,B 0,C 180,E1 33413.38,E2 33413.38} C_VEL
LIN {X 0,Y 713.719,Z 1039.823,A -85,B 0,C 180,E1 33411.961,E2 33411.961} C_VEL
LIN {X 0,Y 713.296,Z 1056.461,A -85,B 0,C 180,E1 33410.515,E2 33410.515} C_VEL
LIN {X 0,Y 712.946,Z 1072.964,A -85,B 0,C 180,E1 33408.903,E2 33408.903} C_VEL
LIN {X 0,Y 712.617,Z 1087.221,A -85,B 0,C 180,E1 33407.305,E2 33407.305} C_VEL
LIN {X 0,Y 712.39,Z 1101.059,A -85,B 0,C 180,E1 33405.55,E2 33405.55} C_VEL
LIN {X 0,Y 712.209,Z 1112.796,A -85,B 0,C 180,E1 33403.808,E2 33403.808} C_VEL
LIN {X 0,Y 712.083,Z 1122.948,A -85,B 0,C 180,E1 33402.077,E2 33402.077} C_VEL
LIN {X 0,Y 711.989,Z 1132.538,A -85,B 0,C 180,E1 33400.11,E2 33400.11} C_VEL
LIN {X 0,Y 711.941,Z 1139.119,A -85,B 0,C 180,E1 33398.48,E2 33398.48} C_VEL
LIN {X 0,Y 711.917,Z 1145.451,A -85,B 0,C 180,E1 33396.532,E2 33396.532} C_VEL
LIN {X 0,Y 711.914,Z 1149.814,A -85,B 0,C 180,E1 33394.673,E2 33394.673} C_VEL
LIN {X 0,Y 711.882,Z 1152.685,A -85,B 0,C 180,E1 33392.898,E2 33392.898} C_VEL
LIN {X 0,Y 711.891,Z 1154.262,A -85,B 0,C 180,E1 33390.885,E2 33390.885} C_VEL
